Yaskawa INFORM job: A_ROOF_UPPER_0614_2_PAINT_55.JBI

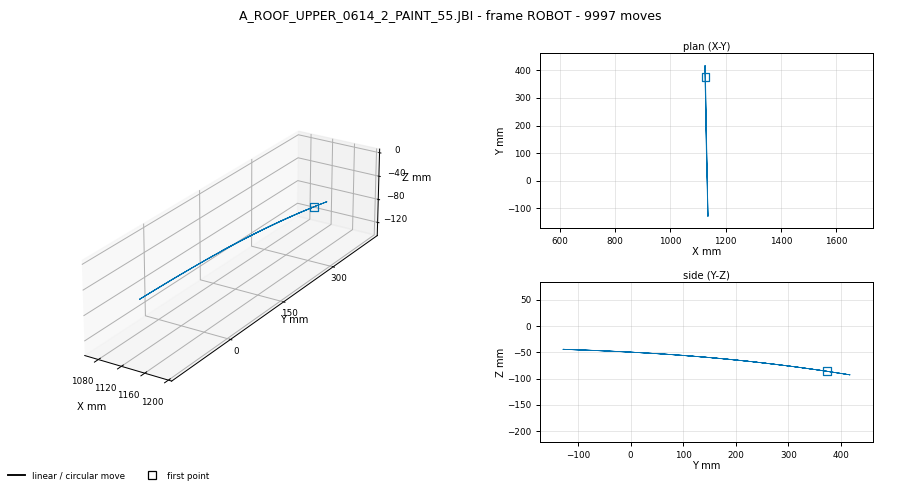
[picture p0: tool path of A_ROOF_UPPER_0614_2_PAINT_55.JBI in frame ROBOT, 9997 of 9997 moves have a stored position in this frame; points joined in program order, loops and branches not executed]
/JOB
//NAME A_ROOF_UPPER_0614_2_PAINT55
//POS
///NPOS 9997,0,0,0,0,0
///TOOL 1
///USER 0
///POSTYPE ROBOT
///RECTAN
///RCONF 1,0,0,0,0,0,0,0,0,0,0,0,0,0,0,0,0,0,0,0,0,0,0,0
C00000=1127.234,374.192,-85.938,-176.955,11.183,149.475
C00001=1127.238,373.945,-85.902,-176.958,11.180,149.475
C00002=1127.242,373.698,-85.865,-176.961,11.179,149.476
C00003=1127.246,373.451,-85.827,-176.964,11.176,149.476
C00004=1127.249,373.204,-85.790,-176.967,11.174,149.476
C00005=1127.253,372.957,-85.754,-176.971,11.171,149.476
C00006=1127.257,372.709,-85.717,-176.973,11.170,149.477
C00007=1127.261,372.462,-85.680,-176.976,11.167,149.477
C00008=1127.264,372.215,-85.643,-176.979,11.164,149.477
C00009=1127.268,371.968,-85.606,-176.983,11.162,149.477
C00010=1127.272,371.720,-85.570,-176.985,11.160,149.477
C00011=1127.276,371.473,-85.533,-176.989,11.158,149.477
C00012=1127.279,371.226,-85.496,-176.992,11.155,149.478
C00013=1127.283,370.978,-85.459,-176.995,11.153,149.478
C00014=1127.287,370.731,-85.423,-176.998,11.151,149.478
C00015=1127.291,370.484,-85.387,-177.001,11.149,149.478
C00016=1127.295,370.236,-85.350,-177.005,11.146,149.479
C00017=1127.299,369.989,-85.313,-177.008,11.144,149.479
C00018=1127.302,369.742,-85.276,-177.011,11.141,149.479
C00019=1127.306,369.495,-85.240,-177.014,11.139,149.479
C00020=1127.310,369.247,-85.203,-177.017,11.137,149.479
C00021=1127.313,369.000,-85.166,-177.020,11.134,149.480
C00022=1127.318,368.753,-85.130,-177.024,11.132,149.480
C00023=1127.321,368.506,-85.094,-177.027,11.130,149.480
C00024=1127.325,368.259,-85.057,-177.030,11.128,149.480
C00025=1127.329,368.011,-85.020,-177.033,11.125,149.480
C00026=1127.332,367.763,-84.984,-177.036,11.123,149.481
C00027=1127.336,367.516,-84.948,-177.040,11.120,149.481
C00028=1127.340,367.269,-84.911,-177.043,11.118,149.481
C00029=1127.344,367.022,-84.874,-177.046,11.115,149.481
C00030=1127.348,366.774,-84.839,-177.050,11.113,149.482
C00031=1127.352,366.527,-84.802,-177.053,11.112,149.482
C00032=1127.356,366.280,-84.765,-177.056,11.109,149.482
C00033=1127.359,366.033,-84.730,-177.059,11.107,149.482
C00034=1127.363,365.785,-84.693,-177.063,11.104,149.483
C00035=1127.367,365.538,-84.656,-177.066,11.102,149.483
C00036=1127.371,365.291,-84.620,-177.069,11.099,149.483
C00037=1127.374,365.043,-84.584,-177.072,11.097,149.483
C00038=1127.378,364.795,-84.548,-177.076,11.094,149.483
C00039=1127.382,364.548,-84.511,-177.079,11.092,149.484
C00040=1127.386,364.301,-84.474,-177.082,11.090,149.484
C00041=1127.390,364.054,-84.439,-177.085,11.088,149.484
C00042=1127.393,363.807,-84.403,-177.089,11.086,149.485
C00043=1127.397,363.559,-84.367,-177.092,11.083,149.485
C00044=1127.401,363.312,-84.330,-177.096,11.081,149.485
C00045=1127.405,363.064,-84.294,-177.099,11.078,149.485
C00046=1127.408,362.852,-84.263,-177.102,11.076,149.486
C00047=1127.412,362.640,-84.232,-177.105,11.074,149.486
C00048=1127.415,362.426,-84.201,-177.107,11.072,149.486
C00049=1127.418,362.214,-84.170,-177.111,11.070,149.486
C00050=1127.421,362.001,-84.139,-177.113,11.068,149.486
C00051=1127.425,361.789,-84.108,-177.117,11.066,149.487
C00052=1127.428,361.576,-84.077,-177.119,11.064,149.487
C00053=1127.431,361.363,-84.046,-177.122,11.062,149.487
C00054=1127.435,361.116,-84.010,-177.125,11.060,149.487
C00055=1127.438,360.869,-83.974,-177.129,11.057,149.488
C00056=1127.443,360.621,-83.938,-177.132,11.055,149.488
C00057=1127.446,360.374,-83.902,-177.136,11.052,149.488
C00058=1127.450,360.127,-83.866,-177.140,11.049,149.488
C00059=1127.453,359.879,-83.831,-177.143,11.047,149.489
C00060=1127.458,359.631,-83.795,-177.147,11.045,149.489
C00061=1127.461,359.384,-83.758,-177.150,11.042,149.489
C00062=1127.465,359.137,-83.723,-177.153,11.040,149.489
C00063=1127.470,358.890,-83.687,-177.156,11.037,149.490
C00064=1127.473,358.642,-83.651,-177.160,11.035,149.490
C00065=1127.477,358.395,-83.615,-177.163,11.033,149.490
C00066=1127.480,358.148,-83.580,-177.167,11.030,149.490
C00067=1127.485,357.900,-83.544,-177.170,11.028,149.491
C00068=1127.488,357.653,-83.508,-177.174,11.026,149.491
C00069=1127.492,357.405,-83.472,-177.177,11.023,149.491
C00070=1127.496,357.158,-83.437,-177.180,11.021,149.491
C00071=1127.499,356.910,-83.401,-177.184,11.018,149.492
C00072=1127.504,356.663,-83.364,-177.188,11.015,149.492
C00073=1127.508,356.416,-83.329,-177.191,11.013,149.492
C00074=1127.511,356.169,-83.294,-177.195,11.011,149.493
C00075=1127.515,355.921,-83.258,-177.198,11.008,149.493
C00076=1127.519,355.674,-83.223,-177.202,11.006,149.493
C00077=1127.522,355.426,-83.187,-177.206,11.003,149.493
C00078=1127.526,355.179,-83.152,-177.209,11.000,149.494
C00079=1127.531,354.932,-83.116,-177.212,10.998,149.494
C00080=1127.535,354.684,-83.080,-177.216,10.996,149.494
C00081=1127.538,354.437,-83.045,-177.219,10.993,149.494
C00082=1127.542,354.189,-83.009,-177.223,10.990,149.495
C00083=1127.546,353.941,-82.974,-177.227,10.988,149.495
C00084=1127.550,353.693,-82.939,-177.230,10.985,149.495
C00085=1127.554,353.447,-82.904,-177.233,10.983,149.495
C00086=1127.558,353.199,-82.868,-177.237,10.980,149.496
C00087=1127.561,352.952,-82.832,-177.241,10.978,149.496
C00088=1127.565,352.704,-82.797,-177.244,10.975,149.496
C00089=1127.569,352.457,-82.762,-177.248,10.973,149.497
C00090=1127.573,352.209,-82.727,-177.252,10.969,149.497
C00091=1127.577,351.962,-82.691,-177.255,10.967,149.497
C00092=1127.581,351.714,-82.656,-177.259,10.965,149.497
C00093=1127.585,351.467,-82.621,-177.262,10.962,149.498
C00094=1127.588,351.220,-82.585,-177.266,10.959,149.498
C00095=1127.592,350.972,-82.550,-177.269,10.957,149.498
C00096=1127.596,350.724,-82.515,-177.273,10.954,149.498
C00097=1127.600,350.478,-82.480,-177.277,10.951,149.499
C00098=1127.604,350.229,-82.445,-177.280,10.949,149.499
C00099=1127.608,349.982,-82.409,-177.284,10.946,149.499
C00100=1127.612,349.734,-82.374,-177.287,10.943,149.499
C00101=1127.616,349.487,-82.339,-177.291,10.941,149.500
C00102=1127.619,349.274,-82.309,-177.294,10.938,149.500
C00103=1127.623,349.061,-82.279,-177.297,10.936,149.500
C00104=1127.626,348.848,-82.248,-177.299,10.935,149.500
C00105=1127.629,348.636,-82.219,-177.302,10.932,149.500
C00106=1127.633,348.423,-82.188,-177.305,10.930,149.501
C00107=1127.636,348.210,-82.159,-177.308,10.928,149.501
C00108=1127.639,347.997,-82.128,-177.311,10.926,149.501
C00109=1127.643,347.785,-82.098,-177.313,10.924,149.501
C00110=1127.646,347.537,-82.063,-177.316,10.921,149.501
C00111=1127.651,347.290,-82.028,-177.320,10.919,149.501
C00112=1127.654,347.042,-81.993,-177.323,10.916,149.502
C00113=1127.658,346.794,-81.958,-177.326,10.914,149.502
C00114=1127.663,346.547,-81.923,-177.330,10.912,149.502
C00115=1127.667,346.299,-81.888,-177.333,10.909,149.502
C00116=1127.670,346.052,-81.853,-177.336,10.907,149.502
C00117=1127.674,345.805,-81.819,-177.339,10.904,149.503
C00118=1127.678,345.557,-81.784,-177.342,10.901,149.503
C00119=1127.682,345.310,-81.749,-177.346,10.899,149.503
C00120=1127.686,345.062,-81.714,-177.349,10.896,149.503
C00121=1127.690,344.814,-81.680,-177.352,10.894,149.503
C00122=1127.694,344.567,-81.644,-177.356,10.892,149.504
C00123=1127.698,344.319,-81.610,-177.359,10.889,149.504
C00124=1127.702,344.072,-81.576,-177.362,10.886,149.504
C00125=1127.705,343.824,-81.540,-177.365,10.884,149.504
C00126=1127.710,343.577,-81.506,-177.369,10.881,149.504
C00127=1127.714,343.329,-81.471,-177.372,10.879,149.505
C00128=1127.717,343.082,-81.436,-177.375,10.876,149.505
C00129=1127.721,342.834,-81.401,-177.378,10.874,149.505
C00130=1127.725,342.586,-81.367,-177.381,10.871,149.505
C00131=1127.729,342.339,-81.333,-177.385,10.869,149.505
C00132=1127.733,342.091,-81.298,-177.388,10.866,149.506
C00133=1127.737,341.844,-81.263,-177.391,10.865,149.506
C00134=1127.741,341.596,-81.228,-177.394,10.862,149.506
C00135=1127.745,341.349,-81.194,-177.397,10.860,149.506
C00136=1127.749,341.101,-81.159,-177.400,10.857,149.506
C00137=1127.753,340.854,-81.125,-177.404,10.854,149.507
C00138=1127.757,340.605,-81.090,-177.407,10.852,149.507
C00139=1127.761,340.358,-81.057,-177.410,10.850,149.507
C00140=1127.765,340.110,-81.022,-177.413,10.847,149.507
C00141=1127.769,339.863,-80.987,-177.416,10.844,149.507
C00142=1127.772,339.615,-80.953,-177.420,10.842,149.508
C00143=1127.777,339.368,-80.918,-177.423,10.839,149.508
C00144=1127.781,339.121,-80.884,-177.426,10.837,149.508
C00145=1127.785,338.873,-80.849,-177.430,10.835,149.508
C00146=1127.788,338.626,-80.815,-177.433,10.832,149.508
C00147=1127.793,338.377,-80.781,-177.436,10.829,149.509
C00148=1127.797,338.130,-80.747,-177.439,10.827,149.509
C00149=1127.800,337.882,-80.712,-177.443,10.824,149.509
C00150=1127.805,337.635,-80.678,-177.445,10.822,149.509
C00151=1127.808,337.387,-80.644,-177.449,10.819,149.509
C00152=1127.812,337.140,-80.610,-177.452,10.817,149.510
C00153=1127.817,336.892,-80.575,-177.455,10.814,149.510
C00154=1127.820,336.644,-80.541,-177.459,10.812,149.510
C00155=1127.824,336.397,-80.507,-177.462,10.809,149.510
C00156=1127.828,336.149,-80.472,-177.464,10.807,149.510
C00157=1127.832,335.902,-80.438,-177.468,10.805,149.511
C00158=1127.836,335.689,-80.409,-177.471,10.802,149.511
C00159=1127.839,335.475,-80.380,-177.473,10.800,149.511
C00160=1127.842,335.262,-80.351,-177.476,10.798,149.511
C00161=1127.845,335.050,-80.321,-177.479,10.796,149.511
C00162=1127.850,334.837,-80.292,-177.481,10.794,149.511
C00163=1127.853,334.623,-80.263,-177.484,10.792,149.512
C00164=1127.856,334.411,-80.233,-177.487,10.790,149.512
C00165=1127.859,334.198,-80.204,-177.490,10.787,149.512
C00166=1127.863,333.950,-80.170,-177.493,10.785,149.512
C00167=1127.867,333.702,-80.136,-177.497,10.782,149.512
C00168=1127.871,333.455,-80.102,-177.499,10.780,149.513
C00169=1127.875,333.207,-80.068,-177.502,10.778,149.513
C00170=1127.879,332.959,-80.034,-177.506,10.775,149.513
C00171=1127.883,332.712,-80.000,-177.509,10.773,149.513
C00172=1127.886,332.464,-79.966,-177.512,10.770,149.513
C00173=1127.891,332.216,-79.932,-177.515,10.768,149.514
C00174=1127.895,331.969,-79.899,-177.519,10.765,149.514
C00175=1127.898,331.721,-79.864,-177.521,10.762,149.514
C00176=1127.903,331.473,-79.831,-177.525,10.760,149.514
C00177=1127.907,331.226,-79.797,-177.528,10.757,149.514
C00178=1127.911,330.979,-79.764,-177.531,10.755,149.515
C00179=1127.914,330.731,-79.729,-177.534,10.752,149.515
C00180=1127.919,330.483,-79.696,-177.538,10.750,149.515
C00181=1127.923,330.236,-79.662,-177.541,10.747,149.515
C00182=1127.927,329.987,-79.628,-177.544,10.745,149.515
C00183=1127.931,329.740,-79.594,-177.547,10.742,149.515
C00184=1127.935,329.492,-79.561,-177.551,10.740,149.516
C00185=1127.939,329.245,-79.527,-177.554,10.737,149.516
C00186=1127.943,328.997,-79.493,-177.557,10.734,149.516
C00187=1127.947,328.749,-79.460,-177.560,10.732,149.516
C00188=1127.951,328.502,-79.426,-177.563,10.730,149.517
C00189=1127.955,328.254,-79.393,-177.566,10.728,149.517
C00190=1127.958,328.006,-79.359,-177.569,10.725,149.517
C00191=1127.963,327.758,-79.325,-177.572,10.723,149.517
C00192=1127.967,327.510,-79.292,-177.576,10.720,149.517
C00193=1127.971,327.263,-79.258,-177.579,10.717,149.517
C00194=1127.975,327.016,-79.225,-177.582,10.715,149.518
C00195=1127.979,326.767,-79.191,-177.585,10.713,149.518
C00196=1127.983,326.520,-79.157,-177.588,10.710,149.518
C00197=1127.987,326.272,-79.124,-177.592,10.707,149.518
C00198=1127.991,326.025,-79.091,-177.595,10.705,149.518
C00199=1127.995,325.777,-79.058,-177.598,10.702,149.518
C00200=1127.999,325.530,-79.024,-177.601,10.700,149.519
C00201=1128.002,325.281,-78.991,-177.604,10.697,149.519
C00202=1128.006,325.034,-78.957,-177.608,10.695,149.519
C00203=1128.011,324.786,-78.924,-177.611,10.692,149.519
C00204=1128.015,324.538,-78.891,-177.614,10.690,149.520
C00205=1128.019,324.291,-78.857,-177.617,10.687,149.520
C00206=1128.023,324.043,-78.824,-177.620,10.684,149.520
C00207=1128.027,323.795,-78.790,-177.624,10.682,149.520
C00208=1128.030,323.547,-78.757,-177.626,10.680,149.520
C00209=1128.034,323.299,-78.724,-177.629,10.677,149.520
C00210=1128.039,323.052,-78.691,-177.633,10.675,149.521
C00211=1128.043,322.804,-78.658,-177.636,10.673,149.521
C00212=1128.047,322.556,-78.625,-177.639,10.670,149.521
C00213=1128.051,322.308,-78.592,-177.642,10.667,149.521
C00214=1128.055,322.096,-78.563,-177.645,10.665,149.521
C00215=1128.058,321.883,-78.534,-177.648,10.663,149.522
C00216=1128.062,321.669,-78.506,-177.650,10.661,149.522
C00217=1128.064,321.456,-78.477,-177.653,10.658,149.522
C00218=1128.068,321.243,-78.448,-177.656,10.656,149.522
C00219=1128.071,321.030,-78.420,-177.659,10.654,149.522
C00220=1128.075,320.817,-78.391,-177.661,10.652,149.522
C00221=1128.078,320.603,-78.364,-177.664,10.650,149.522
C00222=1128.082,320.356,-78.330,-177.667,10.648,149.523
C00223=1128.086,320.108,-78.297,-177.670,10.645,149.523
C00224=1128.090,319.860,-78.264,-177.673,10.642,149.523
C00225=1128.095,319.613,-78.231,-177.676,10.640,149.523
C00226=1128.099,319.365,-78.198,-177.680,10.637,149.524
C00227=1128.102,319.117,-78.165,-177.683,10.635,149.524
C00228=1128.106,318.870,-78.132,-177.686,10.632,149.524
C00229=1128.111,318.621,-78.100,-177.689,10.629,149.524
C00230=1128.115,318.374,-78.066,-177.692,10.627,149.524
C00231=1128.119,318.126,-78.033,-177.696,10.625,149.524
C00232=1128.122,317.878,-78.001,-177.699,10.622,149.525
C00233=1128.127,317.631,-77.968,-177.702,10.619,149.525
C00234=1128.131,317.382,-77.935,-177.705,10.617,149.525
C00235=1128.135,317.135,-77.902,-177.708,10.614,149.525
C00236=1128.139,316.887,-77.869,-177.711,10.613,149.525
C00237=1128.143,316.639,-77.836,-177.714,10.610,149.525
C00238=1128.147,316.391,-77.804,-177.717,10.607,149.526
C00239=1128.151,316.144,-77.771,-177.720,10.605,149.526
C00240=1128.155,315.896,-77.738,-177.723,10.602,149.526
C00241=1128.159,315.648,-77.706,-177.727,10.600,149.526
C00242=1128.163,315.400,-77.673,-177.730,10.597,149.527
C00243=1128.167,315.152,-77.640,-177.733,10.594,149.527
C00244=1128.171,314.904,-77.608,-177.736,10.592,149.527
C00245=1128.175,314.656,-77.574,-177.739,10.589,149.527
C00246=1128.179,314.408,-77.543,-177.742,10.587,149.527
C00247=1128.183,314.161,-77.509,-177.746,10.584,149.527
C00248=1128.187,313.913,-77.476,-177.749,10.582,149.528
C00249=1128.191,313.665,-77.444,-177.752,10.579,149.528
C00250=1128.196,313.418,-77.412,-177.755,10.576,149.528
C00251=1128.199,313.170,-77.380,-177.758,10.574,149.528
C00252=1128.203,312.922,-77.347,-177.761,10.572,149.528
C00253=1128.208,312.674,-77.314,-177.764,10.569,149.528
C00254=1128.211,312.426,-77.282,-177.767,10.567,149.529
C00255=1128.216,312.178,-77.249,-177.770,10.564,149.529
C00256=1128.219,311.931,-77.217,-177.774,10.562,149.529
C00257=1128.224,311.682,-77.184,-177.777,10.559,149.529
C00258=1128.228,311.435,-77.153,-177.780,10.557,149.529
C00259=1128.232,311.187,-77.119,-177.783,10.554,149.530
C00260=1128.236,310.939,-77.087,-177.786,10.551,149.530
C00261=1128.240,310.691,-77.054,-177.789,10.549,149.530
C00262=1128.244,310.443,-77.022,-177.792,10.546,149.530
C00263=1128.248,310.195,-76.990,-177.796,10.544,149.530
C00264=1128.252,309.947,-76.957,-177.799,10.541,149.531
C00265=1128.256,309.700,-76.926,-177.802,10.539,149.531
C00266=1128.261,309.452,-76.893,-177.805,10.536,149.531
C00267=1128.264,309.204,-76.861,-177.808,10.533,149.531
C00268=1128.269,308.956,-76.828,-177.811,10.532,149.531
C00269=1128.272,308.708,-76.796,-177.814,10.529,149.531
C00270=1128.276,308.495,-76.769,-177.817,10.527,149.532
C00271=1128.280,308.282,-76.741,-177.819,10.525,149.532
C00272=1128.283,308.069,-76.713,-177.822,10.522,149.532
C00273=1128.287,307.855,-76.685,-177.825,10.520,149.532
C00274=1128.290,307.642,-76.658,-177.827,10.518,149.532
C00275=1128.293,307.429,-76.630,-177.831,10.516,149.532
C00276=1128.298,307.216,-76.602,-177.833,10.514,149.533
C00277=1128.301,307.002,-76.575,-177.835,10.512,149.533
C00278=1128.305,306.754,-76.542,-177.839,10.509,149.533
C00279=1128.309,306.506,-76.510,-177.842,10.506,149.533
C00280=1128.313,306.259,-76.479,-177.845,10.504,149.533
C00281=1128.318,306.011,-76.446,-177.848,10.501,149.533
C00282=1128.321,305.763,-76.415,-177.851,10.499,149.534
C00283=1128.325,305.514,-76.383,-177.854,10.496,149.534
C00284=1128.330,305.267,-76.351,-177.857,10.494,149.534
C00285=1128.334,305.019,-76.319,-177.861,10.491,149.534
C00286=1128.337,304.771,-76.287,-177.864,10.488,149.534
C00287=1128.342,304.523,-76.255,-177.867,10.486,149.535
C00288=1128.346,304.275,-76.223,-177.870,10.483,149.535
C00289=1128.350,304.027,-76.191,-177.873,10.481,149.535
C00290=1128.354,303.779,-76.159,-177.876,10.478,149.535
C00291=1128.359,303.531,-76.127,-177.879,10.476,149.535
C00292=1128.362,303.283,-76.095,-177.882,10.474,149.535
C00293=1128.366,303.035,-76.064,-177.885,10.471,149.536
C00294=1128.371,302.788,-76.032,-177.888,10.468,149.536
C00295=1128.375,302.540,-76.000,-177.891,10.466,149.536
C00296=1128.378,302.292,-75.968,-177.894,10.463,149.536
C00297=1128.383,302.044,-75.936,-177.898,10.461,149.536
C00298=1128.387,301.796,-75.904,-177.901,10.458,149.537
C00299=1128.392,301.549,-75.872,-177.904,10.456,149.537
C00300=1128.396,301.300,-75.841,-177.907,10.453,149.537
C00301=1128.399,301.052,-75.809,-177.910,10.450,149.537
C00302=1128.404,300.805,-75.778,-177.914,10.448,149.537
C00303=1128.408,300.556,-75.746,-177.916,10.445,149.537
C00304=1128.412,300.308,-75.714,-177.919,10.444,149.538
C00305=1128.416,300.060,-75.683,-177.922,10.441,149.538
C00306=1128.420,299.812,-75.651,-177.925,10.438,149.538
C00307=1128.424,299.565,-75.620,-177.928,10.436,149.538
C00308=1128.428,299.317,-75.588,-177.932,10.433,149.538
C00309=1128.432,299.068,-75.557,-177.935,10.430,149.538
C00310=1128.437,298.820,-75.525,-177.938,10.428,149.539
C00311=1128.441,298.572,-75.493,-177.941,10.425,149.539
C00312=1128.445,298.324,-75.462,-177.944,10.423,149.539
C00313=1128.449,298.076,-75.430,-177.947,10.420,149.539
C00314=1128.453,297.829,-75.399,-177.951,10.418,149.539
C00315=1128.457,297.580,-75.367,-177.953,10.415,149.540
C00316=1128.461,297.332,-75.336,-177.957,10.412,149.540
C00317=1128.465,297.085,-75.304,-177.959,10.410,149.540
C00318=1128.469,296.836,-75.273,-177.962,10.408,149.540
C00319=1128.474,296.589,-75.242,-177.965,10.405,149.540
C00320=1128.478,296.340,-75.210,-177.969,10.403,149.541
C00321=1128.482,296.093,-75.179,-177.972,10.400,149.541
C00322=1128.486,295.844,-75.148,-177.975,10.398,149.541
C00323=1128.490,295.597,-75.116,-177.978,10.395,149.541
C00324=1128.494,295.348,-75.085,-177.981,10.392,149.541
C00325=1128.499,295.101,-75.054,-177.984,10.390,149.541
C00326=1128.502,294.887,-75.027,-177.986,10.388,149.541
C00327=1128.506,294.673,-75.000,-177.990,10.385,149.542
C00328=1128.509,294.461,-74.973,-177.992,10.383,149.542
C00329=1128.513,294.247,-74.946,-177.994,10.381,149.542
C00330=1128.517,294.034,-74.919,-177.998,10.379,149.542
C00331=1128.520,293.820,-74.893,-178.000,10.377,149.542
C00332=1128.523,293.607,-74.865,-178.002,10.375,149.542
C00333=1128.527,293.394,-74.839,-178.005,10.372,149.542
C00334=1128.531,293.145,-74.807,-178.009,10.370,149.543
C00335=1128.536,292.897,-74.777,-178.012,10.367,149.543
C00336=1128.539,292.649,-74.745,-178.015,10.364,149.543
C00337=1128.543,292.402,-74.715,-178.017,10.362,149.543
C00338=1128.547,292.154,-74.683,-178.021,10.360,149.544
C00339=1128.552,291.906,-74.652,-178.023,10.357,149.544
C00340=1128.556,291.658,-74.621,-178.027,10.355,149.544
C00341=1128.560,291.409,-74.590,-178.030,10.352,149.544
C00342=1128.565,291.162,-74.559,-178.033,10.350,149.544
C00343=1128.568,290.913,-74.528,-178.036,10.347,149.544
C00344=1128.572,290.665,-74.497,-178.039,10.345,149.545
C00345=1128.576,290.417,-74.466,-178.042,10.342,149.545
C00346=1128.581,290.169,-74.435,-178.045,10.339,149.545
C00347=1128.585,289.921,-74.404,-178.049,10.337,149.545
C00348=1128.589,289.673,-74.373,-178.051,10.335,149.545
C00349=1128.593,289.425,-74.343,-178.054,10.332,149.545
C00350=1128.597,289.176,-74.312,-178.057,10.329,149.546
C00351=1128.602,288.929,-74.280,-178.060,10.327,149.546
C00352=1128.605,288.681,-74.250,-178.063,10.324,149.546
C00353=1128.609,288.433,-74.219,-178.067,10.322,149.546
C00354=1128.614,288.185,-74.188,-178.070,10.319,149.546
C00355=1128.619,287.937,-74.157,-178.073,10.317,149.547
C00356=1128.622,287.688,-74.127,-178.076,10.314,149.547
C00357=1128.627,287.441,-74.096,-178.079,10.311,149.547
C00358=1128.631,287.193,-74.065,-178.082,10.309,149.547
C00359=1128.634,286.944,-74.035,-178.085,10.307,149.547
C00360=1128.639,286.696,-74.004,-178.088,10.304,149.547
C00361=1128.644,286.448,-73.973,-178.091,10.301,149.548
C00362=1128.647,286.200,-73.943,-178.094,10.299,149.548
C00363=1128.652,285.952,-73.912,-178.097,10.296,149.548
C00364=1128.656,285.704,-73.881,-178.100,10.294,149.548
C00365=1128.659,285.456,-73.851,-178.103,10.291,149.548
C00366=1128.664,285.208,-73.820,-178.106,10.288,149.548
C00367=1128.668,284.960,-73.790,-178.110,10.286,149.549
C00368=1128.673,284.712,-73.759,-178.113,10.283,149.549
C00369=1128.677,284.463,-73.728,-178.115,10.282,149.549
C00370=1128.680,284.216,-73.698,-178.118,10.279,149.549
C00371=1128.685,283.968,-73.667,-178.122,10.276,149.549
C00372=1128.689,283.719,-73.637,-178.125,10.274,149.550
C00373=1128.693,283.471,-73.606,-178.127,10.271,149.550
C00374=1128.698,283.223,-73.575,-178.131,10.268,149.550
C00375=1128.702,282.975,-73.545,-178.134,10.266,149.550
C00376=1128.706,282.727,-73.514,-178.137,10.263,149.550
C00377=1128.710,282.478,-73.485,-178.140,10.260,149.550
C00378=1128.715,282.230,-73.454,-178.143,10.258,149.551
C00379=1128.718,281.983,-73.424,-178.146,10.256,149.551
C00380=1128.723,281.735,-73.393,-178.149,10.253,149.551
C00381=1128.727,281.486,-73.363,-178.152,10.251,149.551
C00382=1128.731,281.273,-73.337,-178.155,10.248,149.551
C00383=1128.734,281.060,-73.311,-178.158,10.246,149.552
C00384=1128.738,280.846,-73.285,-178.161,10.243,149.552
C00385=1128.742,280.632,-73.258,-178.165,10.241,149.552
C00386=1128.745,280.419,-73.233,-178.167,10.239,149.552
C00387=1128.749,280.205,-73.206,-178.170,10.236,149.552
C00388=1128.752,279.992,-73.181,-178.173,10.233,149.552
C00389=1128.756,279.778,-73.154,-178.176,10.231,149.553
C00390=1128.760,279.530,-73.125,-178.179,10.228,149.553
C00391=1128.764,279.282,-73.094,-178.183,10.226,149.553
C00392=1128.768,279.033,-73.064,-178.187,10.223,149.553
C00393=1128.773,278.785,-73.034,-178.190,10.220,149.553
C00394=1128.777,278.538,-73.003,-178.193,10.217,149.554
C00395=1128.781,278.290,-72.974,-178.197,10.214,149.554
C00396=1128.785,278.041,-72.943,-178.200,10.212,149.554
C00397=1128.789,277.793,-72.913,-178.203,10.209,149.554
C00398=1128.793,277.545,-72.883,-178.207,10.206,149.554
C00399=1128.798,277.296,-72.853,-178.210,10.203,149.555
C00400=1128.802,277.049,-72.823,-178.213,10.200,149.555
C00401=1128.806,276.800,-72.794,-178.216,10.198,149.555
C00402=1128.810,276.552,-72.764,-178.219,10.195,149.555
C00403=1128.815,276.304,-72.733,-178.223,10.192,149.555
C00404=1128.819,276.056,-72.704,-178.226,10.189,149.555
C00405=1128.822,275.808,-72.673,-178.229,10.186,149.555
C00406=1128.827,275.559,-72.644,-178.232,10.184,149.556
C00407=1128.832,275.311,-72.614,-178.235,10.181,149.556
C00408=1128.835,275.063,-72.584,-178.238,10.178,149.556
C00409=1128.840,274.815,-72.554,-178.241,10.175,149.556
C00410=1128.844,274.567,-72.525,-178.244,10.173,149.556
C00411=1128.848,274.319,-72.494,-178.247,10.170,149.556
C00412=1128.853,274.070,-72.465,-178.250,10.168,149.557
C00413=1128.857,273.822,-72.435,-178.253,10.165,149.557
C00414=1128.861,273.574,-72.406,-178.256,10.162,149.557
C00415=1128.865,273.326,-72.375,-178.259,10.160,149.557
C00416=1128.869,273.078,-72.346,-178.262,10.157,149.557
C00417=1128.874,272.829,-72.316,-178.265,10.154,149.557
C00418=1128.878,272.581,-72.287,-178.268,10.151,149.557
C00419=1128.882,272.333,-72.257,-178.271,10.149,149.557
C00420=1128.886,272.085,-72.227,-178.274,10.146,149.558
C00421=1128.890,271.837,-72.197,-178.277,10.143,149.558
C00422=1128.895,271.589,-72.168,-178.280,10.140,149.558
C00423=1128.899,271.340,-72.139,-178.283,10.138,149.558
C00424=1128.903,271.092,-72.109,-178.285,10.136,149.558
C00425=1128.908,270.844,-72.079,-178.288,10.133,149.558
C00426=1128.912,270.595,-72.050,-178.292,10.130,149.558
C00427=1128.916,270.347,-72.020,-178.295,10.128,149.558
C00428=1128.920,270.099,-71.991,-178.297,10.125,149.559
C00429=1128.924,269.851,-71.961,-178.299,10.123,149.559
C00430=1128.928,269.603,-71.931,-178.302,10.120,149.559
C00431=1128.933,269.355,-71.902,-178.305,10.117,149.559
C00432=1128.937,269.106,-71.872,-178.308,10.115,149.559
C00433=1128.941,268.858,-71.843,-178.310,10.112,149.559
C00434=1128.946,268.610,-71.814,-178.313,10.110,149.559
C00435=1128.950,268.362,-71.784,-178.316,10.108,149.559
C00436=1128.954,268.113,-71.755,-178.319,10.105,149.559
C00437=1128.959,267.865,-71.726,-178.321,10.103,149.559
C00438=1128.962,267.652,-71.701,-178.324,10.100,149.560
C00439=1128.966,267.438,-71.676,-178.326,10.098,149.560
C00440=1128.969,267.224,-71.649,-178.328,10.096,149.560
C00441=1128.973,267.010,-71.624,-178.330,10.094,149.560
C00442=1128.977,266.797,-71.599,-178.333,10.092,149.560
C00443=1128.980,266.583,-71.574,-178.335,10.090,149.560
C00444=1128.984,266.369,-71.549,-178.337,10.087,149.560
C00445=1128.988,266.156,-71.524,-178.339,10.085,149.560
C00446=1128.992,265.908,-71.495,-178.342,10.084,149.560
C00447=1128.996,265.659,-71.465,-178.344,10.082,149.560
C00448=1129.000,265.411,-71.436,-178.347,10.079,149.560
C00449=1129.004,265.163,-71.406,-178.349,10.076,149.560
C00450=1129.009,264.914,-71.378,-178.352,10.074,149.560
C00451=1129.014,264.666,-71.349,-178.354,10.072,149.561
C00452=1129.018,264.418,-71.319,-178.356,10.070,149.561
C00453=1129.022,264.170,-71.290,-178.360,10.067,149.561
C00454=1129.026,263.921,-71.261,-178.364,10.063,149.561
C00455=1129.030,263.673,-71.232,-178.368,10.060,149.562
C00456=1129.035,263.426,-71.203,-178.372,10.057,149.562
C00457=1129.039,263.177,-71.174,-178.376,10.053,149.562
C00458=1129.043,262.928,-71.145,-178.380,10.050,149.562
C00459=1129.047,262.680,-71.115,-178.383,10.048,149.562
C00460=1129.052,262.432,-71.086,-178.387,10.044,149.563
C00461=1129.056,262.184,-71.058,-178.391,10.041,149.563
C00462=1129.060,261.936,-71.029,-178.394,10.038,149.563
C00463=1129.065,261.687,-71.000,-178.398,10.035,149.563
C00464=1129.069,261.439,-70.971,-178.401,10.032,149.563
C00465=1129.073,261.191,-70.942,-178.405,10.029,149.564
C00466=1129.077,260.942,-70.913,-178.408,10.026,149.564
C00467=1129.082,260.694,-70.884,-178.411,10.023,149.564
C00468=1129.086,260.445,-70.855,-178.415,10.020,149.564
C00469=1129.090,260.198,-70.827,-178.419,10.016,149.564
C00470=1129.095,259.949,-70.798,-178.422,10.014,149.564
C00471=1129.099,259.701,-70.768,-178.425,10.011,149.565
C00472=1129.103,259.452,-70.740,-178.428,10.008,149.565
C00473=1129.108,259.204,-70.712,-178.431,10.005,149.565
C00474=1129.112,258.956,-70.682,-178.435,10.001,149.565
C00475=1129.116,258.707,-70.654,-178.438,9.999,149.565
C00476=1129.120,258.460,-70.625,-178.441,9.996,149.565
C00477=1129.125,258.211,-70.596,-178.444,9.993,149.565
C00478=1129.129,257.962,-70.568,-178.447,9.990,149.565
C00479=1129.133,257.715,-70.539,-178.450,9.987,149.565
C00480=1129.137,257.466,-70.511,-178.453,9.984,149.566
C00481=1129.142,257.217,-70.482,-178.456,9.981,149.566
C00482=1129.146,256.970,-70.453,-178.459,9.979,149.566
C00483=1129.150,256.721,-70.425,-178.462,9.976,149.566
C00484=1129.155,256.472,-70.396,-178.465,9.973,149.566
C00485=1129.159,256.225,-70.368,-178.468,9.970,149.566
C00486=1129.163,255.976,-70.339,-178.471,9.967,149.566
C00487=1129.167,255.727,-70.311,-178.471,9.966,149.566
C00488=1129.172,255.479,-70.283,-178.470,9.965,149.565
C00489=1129.175,255.231,-70.254,-178.469,9.965,149.565
C00490=1129.181,254.983,-70.225,-178.469,9.963,149.565
C00491=1129.184,254.735,-70.197,-178.470,9.962,149.565
C00492=1129.189,254.486,-70.169,-178.470,9.961,149.564
C00493=1129.194,254.237,-70.140,-178.470,9.960,149.564
C00494=1129.197,254.024,-70.116,-178.472,9.959,149.564
C00495=1129.201,253.810,-70.091,-178.472,9.958,149.564
C00496=1129.204,253.596,-70.067,-178.474,9.957,149.564
C00497=1129.208,253.382,-70.042,-178.475,9.955,149.564
C00498=1129.212,253.169,-70.017,-178.476,9.953,149.564
C00499=1129.215,252.955,-69.993,-178.478,9.951,149.564
C00500=1129.219,252.741,-69.969,-178.480,9.950,149.564
C00501=1129.223,252.527,-69.944,-178.482,9.948,149.564
C00502=1129.227,252.280,-69.916,-178.485,9.945,149.564
C00503=1129.231,252.031,-69.887,-178.488,9.944,149.565
C00504=1129.235,251.782,-69.859,-178.491,9.941,149.565
C00505=1129.240,251.534,-69.830,-178.495,9.938,149.565
C00506=1129.244,251.285,-69.802,-178.497,9.935,149.565
C00507=1129.249,251.037,-69.774,-178.501,9.932,149.566
C00508=1129.253,250.789,-69.746,-178.506,9.929,149.566
C00509=1129.258,250.541,-69.717,-178.511,9.925,149.566
C00510=1129.262,250.292,-69.689,-178.515,9.922,149.567
C00511=1129.265,250.043,-69.661,-178.520,9.918,149.567
C00512=1129.270,249.795,-69.633,-178.525,9.914,149.568
C00513=1129.274,249.547,-69.605,-178.530,9.910,149.568
C00514=1129.279,249.298,-69.576,-178.536,9.905,149.568
C00515=1129.283,249.050,-69.548,-178.541,9.901,149.569
C00516=1129.287,248.802,-69.520,-178.548,9.896,149.569
C00517=1129.291,248.553,-69.492,-178.554,9.892,149.570
C00518=1129.296,248.305,-69.464,-178.560,9.887,149.570
C00519=1129.300,248.057,-69.436,-178.567,9.881,149.571
C00520=1129.305,247.808,-69.409,-178.574,9.876,149.572
C00521=1129.309,247.560,-69.381,-178.581,9.871,149.572
C00522=1129.313,247.311,-69.352,-178.586,9.867,149.572
C00523=1129.318,247.063,-69.324,-178.587,9.864,149.572
C00524=1129.322,246.814,-69.297,-178.588,9.862,149.572
C00525=1129.326,246.566,-69.269,-178.589,9.860,149.572
C00526=1129.330,246.319,-69.241,-178.591,9.858,149.571
C00527=1129.335,246.069,-69.213,-178.592,9.856,149.571
C00528=1129.340,245.821,-69.186,-178.593,9.854,149.571
C00529=1129.343,245.573,-69.157,-178.595,9.852,149.571
C00530=1129.348,245.324,-69.130,-178.596,9.849,149.571
C00531=1129.352,245.076,-69.103,-178.597,9.848,149.571
C00532=1129.356,244.828,-69.074,-178.599,9.845,149.571
C00533=1129.362,244.579,-69.047,-178.601,9.843,149.571
C00534=1129.365,244.330,-69.019,-178.602,9.841,149.570
C00535=1129.370,244.082,-68.991,-178.604,9.839,149.570
C00536=1129.374,243.834,-68.964,-178.606,9.836,149.570
C00537=1129.378,243.585,-68.936,-178.608,9.834,149.570
C00538=1129.383,243.337,-68.909,-178.609,9.833,149.570
C00539=1129.387,243.089,-68.881,-178.611,9.830,149.570
C00540=1129.391,242.840,-68.853,-178.613,9.828,149.570
C00541=1129.396,242.592,-68.825,-178.615,9.826,149.570
C00542=1129.400,242.343,-68.797,-178.617,9.823,149.570
C00543=1129.405,242.094,-68.770,-178.618,9.821,149.570
C00544=1129.409,241.847,-68.742,-178.621,9.819,149.570
C00545=1129.413,241.597,-68.715,-178.623,9.817,149.570
C00546=1129.417,241.350,-68.687,-178.625,9.814,149.570
C00547=1129.422,241.101,-68.660,-178.626,9.812,149.570
C00548=1129.426,240.852,-68.632,-178.629,9.809,149.570
C00549=1129.430,240.604,-68.605,-178.631,9.807,149.570
C00550=1129.434,240.390,-68.581,-178.634,9.805,149.570
C00551=1129.438,240.176,-68.557,-178.635,9.803,149.570
C00552=1129.441,239.963,-68.533,-178.637,9.801,149.570
C00553=1129.446,239.748,-68.510,-178.639,9.799,149.570
C00554=1129.449,239.535,-68.486,-178.641,9.797,149.570
C00555=1129.453,239.321,-68.462,-178.643,9.795,149.570
C00556=1129.457,239.106,-68.439,-178.645,9.792,149.570
C00557=1129.460,238.893,-68.415,-178.647,9.790,149.570
C00558=1129.464,238.644,-68.388,-178.650,9.788,149.571
C00559=1129.469,238.396,-68.361,-178.652,9.785,149.570
C00560=1129.473,238.148,-68.333,-178.655,9.783,149.571
C00561=1129.478,237.899,-68.305,-178.658,9.781,149.571
C00562=1129.482,237.650,-68.278,-178.660,9.778,149.571
C00563=1129.487,237.402,-68.251,-178.662,9.776,149.571
C00564=1129.491,237.154,-68.223,-178.665,9.773,149.571
C00565=1129.495,236.905,-68.196,-178.668,9.770,149.571
C00566=1129.500,236.657,-68.168,-178.671,9.767,149.571
C00567=1129.504,236.408,-68.141,-178.674,9.765,149.571
C00568=1129.509,236.160,-68.114,-178.677,9.762,149.571
C00569=1129.514,235.911,-68.087,-178.679,9.759,149.571
C00570=1129.517,235.663,-68.060,-178.682,9.757,149.571
C00571=1129.521,235.414,-68.032,-178.685,9.754,149.572
C00572=1129.526,235.166,-68.005,-178.689,9.750,149.572
C00573=1129.531,234.917,-67.978,-178.691,9.748,149.572
C00574=1129.535,234.668,-67.951,-178.694,9.745,149.572
C00575=1129.539,234.420,-67.923,-178.697,9.742,149.572
C00576=1129.544,234.172,-67.896,-178.701,9.740,149.572
C00577=1129.548,233.924,-67.870,-178.704,9.737,149.573
C00578=1129.552,233.675,-67.843,-178.707,9.734,149.573
C00579=1129.556,233.426,-67.815,-178.710,9.731,149.573
C00580=1129.561,233.178,-67.788,-178.714,9.727,149.573
C00581=1129.565,232.929,-67.762,-178.717,9.725,149.573
C00582=1129.569,232.681,-67.735,-178.720,9.721,149.573
C00583=1129.574,232.432,-67.707,-178.723,9.718,149.573
C00584=1129.579,232.184,-67.680,-178.727,9.715,149.574
C00585=1129.583,231.935,-67.653,-178.730,9.712,149.574
C00586=1129.587,231.686,-67.627,-178.734,9.709,149.574
C00587=1129.591,231.438,-67.599,-178.737,9.705,149.574
C00588=1129.596,231.189,-67.572,-178.740,9.703,149.574
C00589=1129.600,230.941,-67.546,-178.744,9.699,149.574
C00590=1129.605,230.693,-67.519,-178.748,9.696,149.574
C00591=1129.609,230.444,-67.492,-178.751,9.692,149.575
C00592=1129.613,230.196,-67.465,-178.755,9.689,149.575
C00593=1129.618,229.948,-67.438,-178.759,9.686,149.575
C00594=1129.623,229.699,-67.411,-178.763,9.682,149.575
C00595=1129.626,229.451,-67.385,-178.766,9.679,149.575
C00596=1129.631,229.202,-67.358,-178.770,9.675,149.575
C00597=1129.636,228.953,-67.331,-178.774,9.672,149.576
C00598=1129.639,228.704,-67.304,-178.777,9.668,149.576
C00599=1129.644,228.456,-67.277,-178.781,9.665,149.576
C00600=1129.648,228.208,-67.251,-178.785,9.661,149.576
C00601=1129.653,227.959,-67.225,-178.788,9.658,149.576
C00602=1129.657,227.710,-67.198,-178.792,9.654,149.576
C00603=1129.662,227.462,-67.171,-178.795,9.651,149.576
C00604=1129.666,227.213,-67.145,-178.798,9.647,149.576
C00605=1129.670,226.965,-67.118,-178.802,9.643,149.576
C00606=1129.674,226.751,-67.095,-178.805,9.641,149.577
C00607=1129.678,226.537,-67.072,-178.808,9.638,149.577
C00608=1129.682,226.323,-67.050,-178.810,9.635,149.577
C00609=1129.686,226.109,-67.027,-178.813,9.632,149.577
C00610=1129.690,225.894,-67.004,-178.816,9.629,149.577
C00611=1129.694,225.681,-66.982,-178.819,9.626,149.577
C00612=1129.697,225.466,-66.958,-178.821,9.623,149.577
C00613=1129.701,225.253,-66.936,-178.824,9.620,149.577
C00614=1129.705,225.004,-66.910,-178.828,9.617,149.577
C00615=1129.710,224.755,-66.883,-178.830,9.614,149.577
C00616=1129.714,224.507,-66.857,-178.834,9.610,149.577
C00617=1129.718,224.258,-66.831,-178.837,9.607,149.577
C00618=1129.723,224.009,-66.804,-178.840,9.603,149.577
C00619=1129.727,223.761,-66.778,-178.843,9.601,149.577
C00620=1129.732,223.512,-66.751,-178.846,9.597,149.577
C00621=1129.737,223.265,-66.725,-178.848,9.594,149.577
C00622=1129.741,223.016,-66.700,-178.852,9.590,149.577
C00623=1129.746,222.767,-66.673,-178.855,9.587,149.577
C00624=1129.750,222.518,-66.647,-178.857,9.584,149.577
C00625=1129.754,222.270,-66.621,-178.860,9.580,149.577
C00626=1129.759,222.021,-66.594,-178.863,9.577,149.577
C00627=1129.763,221.772,-66.568,-178.865,9.574,149.577
C00628=1129.767,221.524,-66.542,-178.868,9.571,149.577
C00629=1129.772,221.276,-66.516,-178.870,9.568,149.577
C00630=1129.777,221.027,-66.490,-178.874,9.564,149.577
C00631=1129.781,220.778,-66.464,-178.876,9.561,149.577
C00632=1129.785,220.530,-66.438,-178.879,9.558,149.577
C00633=1129.790,220.281,-66.411,-178.881,9.554,149.576
C00634=1129.794,220.032,-66.386,-178.884,9.551,149.576
C00635=1129.799,219.784,-66.360,-178.886,9.548,149.576
C00636=1129.803,219.536,-66.334,-178.889,9.545,149.576
C00637=1129.808,219.287,-66.307,-178.891,9.542,149.576
C00638=1129.812,219.038,-66.282,-178.894,9.539,149.576
C00639=1129.816,218.789,-66.256,-178.896,9.536,149.576
C00640=1129.820,218.540,-66.230,-178.898,9.533,149.576
C00641=1129.825,218.293,-66.204,-178.900,9.530,149.576
C00642=1129.830,218.044,-66.178,-178.903,9.527,149.576
C00643=1129.834,217.795,-66.152,-178.905,9.524,149.576
C00644=1129.838,217.546,-66.126,-178.907,9.521,149.575
C00645=1129.843,217.298,-66.101,-178.909,9.518,149.575
C00646=1129.847,217.049,-66.075,-178.912,9.515,149.575
C00647=1129.851,216.800,-66.049,-178.913,9.512,149.575
C00648=1129.856,216.551,-66.023,-178.916,9.509,149.575
C00649=1129.861,216.302,-65.997,-178.918,9.507,149.575
C00650=1129.865,216.055,-65.971,-178.920,9.503,149.575
C00651=1129.869,215.806,-65.945,-178.922,9.501,149.574
C00652=1129.874,215.557,-65.920,-178.924,9.497,149.574
C00653=1129.878,215.308,-65.894,-178.926,9.495,149.574
C00654=1129.883,215.060,-65.869,-178.928,9.493,149.574
C00655=1129.887,214.812,-65.843,-178.930,9.489,149.574
C00656=1129.891,214.563,-65.817,-178.932,9.487,149.574
C00657=1129.896,214.315,-65.792,-178.933,9.484,149.574
C00658=1129.901,214.066,-65.765,-178.936,9.481,149.574
C00659=1129.905,213.817,-65.740,-178.937,9.478,149.573
C00660=1129.909,213.568,-65.714,-178.939,9.476,149.573
C00661=1129.914,213.320,-65.688,-178.940,9.473,149.573
C00662=1129.917,213.105,-65.667,-178.941,9.471,149.573
C00663=1129.922,212.891,-65.644,-178.943,9.469,149.573
C00664=1129.925,212.677,-65.623,-178.944,9.467,149.572
C00665=1129.930,212.463,-65.601,-178.946,9.465,149.572
C00666=1129.934,212.249,-65.578,-178.947,9.462,149.572
C00667=1129.937,212.034,-65.556,-178.949,9.461,149.572
C00668=1129.941,211.820,-65.534,-178.951,9.458,149.572
C00669=1129.945,211.606,-65.513,-178.951,9.456,149.572
C00670=1129.949,211.357,-65.487,-178.954,9.453,149.572
C00671=1129.954,211.109,-65.462,-178.956,9.451,149.572
C00672=1129.958,210.860,-65.436,-178.958,9.449,149.572
C00673=1129.962,210.612,-65.410,-178.960,9.446,149.572
C00674=1129.967,210.363,-65.385,-178.961,9.443,149.571
C00675=1129.971,210.114,-65.360,-178.963,9.441,149.571
C00676=1129.976,209.865,-65.334,-178.965,9.438,149.571
C00677=1129.980,209.617,-65.309,-178.967,9.436,149.571
C00678=1129.985,209.368,-65.283,-178.970,9.434,149.571
C00679=1129.989,209.119,-65.258,-178.972,9.431,149.571
C00680=1129.994,208.871,-65.232,-178.974,9.428,149.571
C00681=1129.998,208.622,-65.207,-178.977,9.425,149.571
C00682=1130.003,208.374,-65.181,-178.979,9.423,149.571
C00683=1130.007,208.125,-65.156,-178.981,9.420,149.571
C00684=1130.012,207.876,-65.130,-178.983,9.418,149.571
C00685=1130.017,207.628,-65.105,-178.986,9.415,149.571
C00686=1130.020,207.379,-65.080,-178.989,9.412,149.571
C00687=1130.025,207.130,-65.055,-178.991,9.410,149.571
C00688=1130.029,206.882,-65.030,-178.994,9.407,149.572
C00689=1130.034,206.633,-65.004,-178.996,9.404,149.572
C00690=1130.039,206.384,-64.979,-178.999,9.401,149.572
C00691=1130.043,206.135,-64.953,-179.002,9.398,149.572
C00692=1130.048,205.887,-64.928,-179.004,9.396,149.572
C00693=1130.052,205.638,-64.904,-179.007,9.393,149.572
C00694=1130.057,205.390,-64.878,-179.010,9.390,149.572
C00695=1130.061,205.140,-64.853,-179.012,9.387,149.572
C00696=1130.066,204.892,-64.828,-179.015,9.385,149.572
C00697=1130.070,204.643,-64.803,-179.019,9.381,149.572
C00698=1130.074,204.395,-64.778,-179.022,9.378,149.572
C00699=1130.079,204.146,-64.752,-179.024,9.375,149.572
C00700=1130.083,203.897,-64.727,-179.027,9.373,149.573
C00701=1130.088,203.649,-64.702,-179.030,9.370,149.573
C00702=1130.093,203.399,-64.677,-179.034,9.366,149.573
C00703=1130.097,203.152,-64.652,-179.037,9.364,149.573
C00704=1130.101,202.902,-64.627,-179.040,9.361,149.573
C00705=1130.106,202.653,-64.602,-179.043,9.357,149.573
C00706=1130.110,202.405,-64.577,-179.046,9.355,149.573
C00707=1130.115,202.156,-64.552,-179.050,9.351,149.574
C00708=1130.119,201.907,-64.527,-179.053,9.348,149.574
C00709=1130.124,201.659,-64.503,-179.057,9.345,149.574
C00710=1130.129,201.410,-64.478,-179.060,9.341,149.574
C00711=1130.133,201.161,-64.452,-179.063,9.339,149.574
C00712=1130.137,200.913,-64.428,-179.067,9.335,149.574
C00713=1130.142,200.664,-64.403,-179.070,9.331,149.574
C00714=1130.147,200.416,-64.378,-179.074,9.328,149.575
C00715=1130.150,200.166,-64.353,-179.077,9.324,149.575
C00716=1130.156,199.918,-64.329,-179.081,9.321,149.575
C00717=1130.159,199.669,-64.304,-179.085,9.317,149.575
C00718=1130.164,199.454,-64.282,-179.088,9.315,149.575
C00719=1130.167,199.240,-64.261,-179.090,9.312,149.575
C00720=1130.171,199.026,-64.240,-179.094,9.308,149.575
C00721=1130.175,198.812,-64.218,-179.097,9.306,149.576
C00722=1130.179,198.597,-64.198,-179.101,9.302,149.576
C00723=1130.183,198.384,-64.176,-179.104,9.299,149.576
C00724=1130.188,198.169,-64.155,-179.107,9.296,149.576
C00725=1130.191,197.955,-64.134,-179.110,9.293,149.576
C00726=1130.195,197.706,-64.109,-179.114,9.289,149.576
C00727=1130.200,197.457,-64.084,-179.118,9.285,149.576
C00728=1130.205,197.209,-64.060,-179.122,9.281,149.577
C00729=1130.209,196.959,-64.035,-179.126,9.278,149.577
C00730=1130.214,196.711,-64.011,-179.130,9.273,149.577
C00731=1130.218,196.463,-63.987,-179.134,9.270,149.577
C00732=1130.222,196.213,-63.962,-179.137,9.266,149.577
C00733=1130.227,195.965,-63.938,-179.139,9.264,149.577
C00734=1130.232,195.716,-63.913,-179.140,9.261,149.577
C00735=1130.236,195.467,-63.889,-179.142,9.259,149.577
C00736=1130.241,195.218,-63.864,-179.143,9.256,149.576
C00737=1130.245,194.970,-63.840,-179.145,9.253,149.576
C00738=1130.250,194.721,-63.816,-179.147,9.251,149.576
C00739=1130.254,194.472,-63.791,-179.148,9.248,149.576
C00740=1130.259,194.224,-63.767,-179.149,9.246,149.576
C00741=1130.263,193.975,-63.743,-179.151,9.244,149.576
C00742=1130.268,193.726,-63.718,-179.152,9.241,149.575
C00743=1130.272,193.477,-63.694,-179.154,9.239,149.575
C00744=1130.277,193.228,-63.670,-179.156,9.235,149.575
C00745=1130.282,192.980,-63.646,-179.158,9.233,149.575
C00746=1130.286,192.730,-63.621,-179.160,9.231,149.575
C00747=1130.291,192.482,-63.597,-179.162,9.228,149.575
C00748=1130.295,192.233,-63.573,-179.164,9.226,149.575
C00749=1130.299,191.985,-63.549,-179.165,9.223,149.574
C00750=1130.304,191.735,-63.524,-179.167,9.221,149.574
C00751=1130.309,191.486,-63.500,-179.169,9.218,149.574
C00752=1130.313,191.238,-63.476,-179.171,9.215,149.574
C00753=1130.317,190.990,-63.452,-179.173,9.212,149.574
C00754=1130.323,190.741,-63.427,-179.175,9.209,149.574
C00755=1130.327,190.491,-63.404,-179.177,9.207,149.574
C00756=1130.331,190.243,-63.380,-179.179,9.205,149.574
C00757=1130.336,189.994,-63.355,-179.182,9.202,149.574
C00758=1130.341,189.746,-63.331,-179.184,9.199,149.574
C00759=1130.345,189.497,-63.307,-179.186,9.196,149.574
C00760=1130.349,189.247,-63.283,-179.188,9.193,149.574
C00761=1130.354,188.999,-63.258,-179.190,9.190,149.574
C00762=1130.359,188.750,-63.234,-179.192,9.188,149.574
C00763=1130.363,188.501,-63.211,-179.194,9.185,149.574
C00764=1130.368,188.253,-63.187,-179.196,9.183,149.574
C00765=1130.372,188.004,-63.163,-179.199,9.180,149.573
C00766=1130.377,187.754,-63.138,-179.201,9.176,149.573
C00767=1130.381,187.506,-63.114,-179.203,9.174,149.573
C00768=1130.386,187.257,-63.091,-179.206,9.171,149.574
C00769=1130.390,187.009,-63.067,-179.209,9.168,149.573
C00770=1130.395,186.760,-63.043,-179.211,9.165,149.573
C00771=1130.400,186.511,-63.020,-179.213,9.163,149.573
C00772=1130.405,186.262,-62.995,-179.216,9.160,149.573
C00773=1130.409,186.013,-62.971,-179.218,9.157,149.573
C00774=1130.413,185.799,-62.951,-179.220,9.154,149.573
C00775=1130.416,185.584,-62.931,-179.223,9.151,149.573
C00776=1130.420,185.370,-62.910,-179.225,9.149,149.573
C00777=1130.424,185.155,-62.889,-179.228,9.146,149.573
C00778=1130.429,184.941,-62.869,-179.229,9.144,149.573
C00779=1130.433,184.727,-62.848,-179.231,9.141,149.573
C00780=1130.436,184.513,-62.828,-179.234,9.138,149.573
C00781=1130.440,184.298,-62.807,-179.236,9.136,149.573
C00782=1130.445,184.049,-62.784,-179.239,9.132,149.573
C00783=1130.449,183.801,-62.759,-179.242,9.129,149.573
C00784=1130.454,183.552,-62.736,-179.244,9.126,149.573
C00785=1130.458,183.303,-62.712,-179.247,9.124,149.573
C00786=1130.463,183.054,-62.689,-179.250,9.120,149.573
C00787=1130.467,182.805,-62.665,-179.253,9.117,149.573
C00788=1130.472,182.557,-62.641,-179.256,9.114,149.574
C00789=1130.477,182.308,-62.618,-179.259,9.111,149.574
C00790=1130.481,182.059,-62.595,-179.262,9.107,149.573
C00791=1130.486,181.810,-62.570,-179.265,9.104,149.574
C00792=1130.490,181.561,-62.547,-179.267,9.101,149.574
C00793=1130.495,181.312,-62.524,-179.270,9.097,149.574
C00794=1130.499,181.064,-62.500,-179.273,9.094,149.574
C00795=1130.504,180.815,-62.476,-179.276,9.090,149.574
C00796=1130.509,180.566,-62.453,-179.279,9.087,149.574
C00797=1130.514,180.317,-62.430,-179.283,9.084,149.574
C00798=1130.518,180.068,-62.406,-179.286,9.080,149.574
C00799=1130.523,179.819,-62.382,-179.289,9.077,149.574
C00800=1130.527,179.570,-62.359,-179.292,9.073,149.574
C00801=1130.532,179.321,-62.335,-179.295,9.069,149.574
C00802=1130.536,179.072,-62.313,-179.297,9.066,149.574
C00803=1130.540,178.824,-62.289,-179.299,9.064,149.574
C00804=1130.545,178.575,-62.265,-179.302,9.061,149.574
C00805=1130.550,178.326,-62.242,-179.304,9.057,149.573
C00806=1130.554,178.077,-62.219,-179.306,9.055,149.573
C00807=1130.559,177.828,-62.195,-179.308,9.052,149.573
C00808=1130.564,177.579,-62.172,-179.310,9.049,149.573
C00809=1130.568,177.330,-62.149,-179.312,9.046,149.573
C00810=1130.573,177.081,-62.126,-179.314,9.043,149.573
C00811=1130.577,176.832,-62.102,-179.316,9.040,149.573
C00812=1130.582,176.583,-62.079,-179.319,9.037,149.573
C00813=1130.586,176.335,-62.055,-179.321,9.034,149.573
C00814=1130.591,176.087,-62.033,-179.323,9.031,149.573
C00815=1130.596,175.837,-62.009,-179.325,9.028,149.572
C00816=1130.600,175.588,-61.986,-179.328,9.025,149.572
C00817=1130.605,175.339,-61.962,-179.329,9.023,149.572
C00818=1130.609,175.091,-61.940,-179.332,9.019,149.572
C00819=1130.614,174.842,-61.916,-179.334,9.016,149.572
C00820=1130.619,174.592,-61.894,-179.336,9.014,149.572
C00821=1130.623,174.343,-61.870,-179.338,9.011,149.572
C00822=1130.628,174.095,-61.848,-179.341,9.007,149.572
C00823=1130.633,173.846,-61.825,-179.342,9.005,149.572
C00824=1130.637,173.597,-61.801,-179.345,9.002,149.572
C00825=1130.641,173.348,-61.778,-179.347,8.998,149.572
C00826=1130.646,173.099,-61.755,-179.350,8.995,149.571
C00827=1130.651,172.850,-61.732,-179.351,8.993,149.571
C00828=1130.655,172.601,-61.709,-179.354,8.990,149.571
C00829=1130.660,172.353,-61.686,-179.357,8.986,149.571
C00830=1130.664,172.138,-61.666,-179.358,8.984,149.571
C00831=1130.668,171.924,-61.647,-179.360,8.981,149.571
C00832=1130.671,171.709,-61.627,-179.362,8.978,149.571
C00833=1130.676,171.494,-61.607,-179.364,8.976,149.571
C00834=1130.680,171.280,-61.588,-179.366,8.974,149.571
C00835=1130.684,171.065,-61.567,-179.369,8.971,149.571
C00836=1130.688,170.851,-61.548,-179.370,8.968,149.571
C00837=1130.691,170.636,-61.528,-179.372,8.966,149.571
C00838=1130.697,170.388,-61.505,-179.375,8.962,149.571
C00839=1130.702,170.138,-61.483,-179.377,8.959,149.570
C00840=1130.705,169.890,-61.460,-179.379,8.956,149.570
C00841=1130.710,169.641,-61.436,-179.382,8.953,149.570
C00842=1130.714,169.392,-61.414,-179.384,8.950,149.570
C00843=1130.720,169.143,-61.391,-179.386,8.947,149.570
C00844=1130.724,168.894,-61.368,-179.388,8.944,149.570
C00845=1130.728,168.645,-61.345,-179.391,8.941,149.570
C00846=1130.733,168.395,-61.323,-179.393,8.938,149.570
C00847=1130.738,168.147,-61.300,-179.396,8.934,149.570
C00848=1130.743,167.898,-61.277,-179.398,8.931,149.570
C00849=1130.747,167.649,-61.255,-179.400,8.928,149.570
C00850=1130.752,167.401,-61.232,-179.403,8.925,149.570
C00851=1130.757,167.151,-61.210,-179.405,8.922,149.569
C00852=1130.761,166.902,-61.186,-179.408,8.919,149.569
C00853=1130.765,166.654,-61.164,-179.410,8.915,149.569
C00854=1130.771,166.405,-61.141,-179.413,8.912,149.569
C00855=1130.775,166.156,-61.119,-179.415,8.909,149.569
C00856=1130.780,165.906,-61.096,-179.418,8.906,149.569
C00857=1130.784,165.658,-61.074,-179.420,8.902,149.569
C00858=1130.789,165.409,-61.052,-179.422,8.899,149.569
C00859=1130.793,165.160,-61.028,-179.425,8.896,149.569
C00860=1130.798,164.911,-61.006,-179.427,8.893,149.569
C00861=1130.803,164.662,-60.983,-179.430,8.890,149.569
C00862=1130.807,164.413,-60.961,-179.432,8.886,149.569
C00863=1130.812,164.164,-60.939,-179.434,8.883,149.568
C00864=1130.817,163.915,-60.916,-179.437,8.880,149.568
C00865=1130.821,163.666,-60.894,-179.439,8.877,149.568
C00866=1130.826,163.418,-60.872,-179.442,8.874,149.568
C00867=1130.831,163.168,-60.849,-179.444,8.870,149.568
C00868=1130.835,162.920,-60.827,-179.447,8.867,149.568
C00869=1130.839,162.671,-60.805,-179.449,8.864,149.568
C00870=1130.844,162.421,-60.782,-179.452,8.860,149.568
C00871=1130.849,162.173,-60.760,-179.454,8.857,149.568
C00872=1130.853,161.924,-60.737,-179.457,8.854,149.568
C00873=1130.858,161.674,-60.715,-179.459,8.851,149.568
C00874=1130.863,161.426,-60.693,-179.462,8.847,149.568
C00875=1130.867,161.177,-60.670,-179.464,8.844,149.567
C00876=1130.873,160.928,-60.648,-179.467,8.841,149.567
C00877=1130.877,160.679,-60.626,-179.470,8.837,149.567
C00878=1130.882,160.430,-60.604,-179.472,8.834,149.567
C00879=1130.886,160.181,-60.582,-179.474,8.830,149.567
C00880=1130.891,159.932,-60.559,-179.477,8.827,149.567
C00881=1130.896,159.683,-60.537,-179.480,8.823,149.567
C00882=1130.900,159.434,-60.515,-179.482,8.820,149.567
C00883=1130.905,159.185,-60.494,-179.485,8.817,149.567
C00884=1130.909,158.936,-60.471,-179.487,8.814,149.567
C00885=1130.914,158.687,-60.448,-179.490,8.810,149.567
C00886=1130.918,158.472,-60.430,-179.492,8.807,149.567
C00887=1130.922,158.258,-60.411,-179.494,8.804,149.567
C00888=1130.926,158.043,-60.392,-179.497,8.801,149.566
C00889=1130.930,157.828,-60.373,-179.498,8.798,149.566
C00890=1130.934,157.614,-60.354,-179.501,8.795,149.566
C00891=1130.938,157.399,-60.335,-179.503,8.792,149.566
C00892=1130.943,157.185,-60.316,-179.505,8.789,149.566
C00893=1130.946,156.970,-60.297,-179.507,8.786,149.566
C00894=1130.951,156.721,-60.275,-179.510,8.782,149.566
C00895=1130.955,156.472,-60.253,-179.513,8.779,149.566
C00896=1130.960,156.223,-60.231,-179.516,8.775,149.566
C00897=1130.964,155.974,-60.209,-179.518,8.772,149.566
C00898=1130.969,155.725,-60.188,-179.520,8.768,149.565
C00899=1130.974,155.477,-60.166,-179.523,8.764,149.565
C00900=1130.978,155.227,-60.144,-179.526,8.761,149.565
C00901=1130.983,154.979,-60.122,-179.529,8.757,149.565
C00902=1130.988,154.729,-60.100,-179.531,8.754,149.565
C00903=1130.993,154.480,-60.078,-179.534,8.750,149.565
C00904=1130.997,154.231,-60.056,-179.536,8.747,149.565
C00905=1131.002,153.982,-60.034,-179.540,8.743,149.565
C00906=1131.007,153.733,-60.013,-179.542,8.739,149.565
C00907=1131.012,153.484,-59.991,-179.545,8.735,149.565
C00908=1131.017,153.235,-59.970,-179.547,8.732,149.564
C00909=1131.021,152.986,-59.947,-179.550,8.728,149.564
C00910=1131.026,152.737,-59.926,-179.553,8.725,149.564
C00911=1131.031,152.488,-59.904,-179.555,8.721,149.564
C00912=1131.035,152.238,-59.883,-179.558,8.718,149.564
C00913=1131.039,151.990,-59.862,-179.561,8.713,149.564
C00914=1131.044,151.741,-59.840,-179.563,8.710,149.564
C00915=1131.048,151.492,-59.818,-179.566,8.706,149.563
C00916=1131.054,151.243,-59.797,-179.569,8.702,149.563
C00917=1131.058,150.994,-59.775,-179.571,8.699,149.563
C00918=1131.063,150.745,-59.753,-179.574,8.695,149.563
C00919=1131.068,150.496,-59.732,-179.577,8.690,149.563
C00920=1131.073,150.247,-59.711,-179.579,8.687,149.563
C00921=1131.077,149.998,-59.689,-179.582,8.683,149.563
C00922=1131.082,149.748,-59.668,-179.585,8.679,149.563
C00923=1131.086,149.500,-59.646,-179.587,8.676,149.562
C00924=1131.091,149.250,-59.625,-179.590,8.672,149.562
C00925=1131.096,149.001,-59.603,-179.593,8.667,149.562
C00926=1131.101,148.753,-59.582,-179.596,8.664,149.562
C00927=1131.106,148.504,-59.561,-179.598,8.660,149.562
C00928=1131.109,148.255,-59.539,-179.602,8.656,149.562
C00929=1131.115,148.005,-59.518,-179.604,8.652,149.562
C00930=1131.119,147.757,-59.497,-179.607,8.648,149.561
C00931=1131.125,147.507,-59.476,-179.610,8.645,149.561
C00932=1131.129,147.258,-59.454,-179.612,8.640,149.561
C00933=1131.133,147.009,-59.433,-179.615,8.636,149.561
C00934=1131.138,146.760,-59.412,-179.618,8.632,149.561
C00935=1131.143,146.511,-59.391,-179.621,8.628,149.561
C00936=1131.147,146.263,-59.370,-179.623,8.625,149.561
C00937=1131.152,146.013,-59.348,-179.626,8.621,149.560
C00938=1131.157,145.764,-59.327,-179.629,8.616,149.560
C00939=1131.162,145.515,-59.306,-179.631,8.612,149.560
C00940=1131.167,145.266,-59.285,-179.635,8.608,149.560
C00941=1131.172,145.017,-59.264,-179.637,8.604,149.560
C00942=1131.176,144.802,-59.246,-179.639,8.601,149.559
C00943=1131.179,144.587,-59.228,-179.640,8.598,149.559
C00944=1131.184,144.372,-59.209,-179.641,8.595,149.559
C00945=1131.187,144.157,-59.192,-179.642,8.592,149.558
C00946=1131.192,143.943,-59.173,-179.644,8.590,149.558
C00947=1131.195,143.728,-59.155,-179.644,8.587,149.558
C00948=1131.200,143.513,-59.137,-179.646,8.585,149.557
C00949=1131.204,143.299,-59.119,-179.647,8.581,149.557
C00950=1131.208,143.050,-59.098,-179.649,8.578,149.557
C00951=1131.213,142.801,-59.077,-179.650,8.575,149.556
C00952=1131.218,142.552,-59.056,-179.651,8.571,149.556
C00953=1131.223,142.303,-59.035,-179.653,8.568,149.556
C00954=1131.228,142.053,-59.014,-179.654,8.565,149.555
C00955=1131.232,141.804,-58.993,-179.656,8.562,149.555
C00956=1131.237,141.555,-58.972,-179.657,8.559,149.555
C00957=1131.241,141.306,-58.952,-179.658,8.555,149.554
C00958=1131.246,141.057,-58.931,-179.660,8.552,149.554
C00959=1131.251,140.808,-58.910,-179.662,8.548,149.554
C00960=1131.256,140.559,-58.889,-179.663,8.545,149.553
C00961=1131.260,140.310,-58.868,-179.664,8.542,149.553
C00962=1131.265,140.061,-58.847,-179.666,8.539,149.553
C00963=1131.269,139.812,-58.826,-179.667,8.536,149.552
C00964=1131.274,139.562,-58.806,-179.669,8.532,149.552
C00965=1131.279,139.313,-58.785,-179.670,8.529,149.552
C00966=1131.284,139.064,-58.764,-179.672,8.525,149.551
C00967=1131.288,138.815,-58.744,-179.673,8.523,149.551
C00968=1131.293,138.566,-58.722,-179.675,8.519,149.551
C00969=1131.298,138.318,-58.702,-179.676,8.516,149.550
C00970=1131.303,138.068,-58.681,-179.678,8.512,149.550
C00971=1131.307,137.819,-58.660,-179.679,8.509,149.550
C00972=1131.313,137.570,-58.639,-179.682,8.506,149.549
C00973=1131.317,137.321,-58.619,-179.683,8.503,149.549
C00974=1131.322,137.072,-58.598,-179.685,8.499,149.549
C00975=1131.327,136.823,-58.578,-179.686,8.496,149.548
C00976=1131.331,136.574,-58.557,-179.688,8.493,149.548
C00977=1131.336,136.325,-58.536,-179.689,8.490,149.548
C00978=1131.341,136.076,-58.516,-179.691,8.486,149.547
C00979=1131.346,135.826,-58.495,-179.692,8.483,149.547
C00980=1131.350,135.578,-58.475,-179.694,8.480,149.547
C00981=1131.355,135.329,-58.454,-179.695,8.477,149.547
C00982=1131.360,135.079,-58.433,-179.697,8.473,149.546
C00983=1131.364,134.830,-58.413,-179.698,8.470,149.546
C00984=1131.370,134.580,-58.393,-179.700,8.466,149.545
C00985=1131.374,134.332,-58.372,-179.701,8.464,149.545
C00986=1131.379,134.083,-58.352,-179.704,8.460,149.545
C00987=1131.384,133.833,-58.331,-179.705,8.457,149.545
C00988=1131.388,133.584,-58.311,-179.707,8.454,149.544
C00989=1131.393,133.335,-58.290,-179.708,8.451,149.544
C00990=1131.398,133.086,-58.269,-179.710,8.447,149.544
C00991=1131.402,132.837,-58.249,-179.712,8.444,149.543
C00992=1131.407,132.588,-58.229,-179.713,8.440,149.543
C00993=1131.412,132.338,-58.208,-179.715,8.437,149.543
C00994=1131.417,132.089,-58.188,-179.716,8.434,149.543
C00995=1131.421,131.840,-58.168,-179.718,8.430,149.542
C00996=1131.426,131.591,-58.147,-179.719,8.428,149.542
C00997=1131.431,131.342,-58.127,-179.721,8.424,149.542
C00998=1131.435,131.127,-58.109,-179.723,8.421,149.542
C00999=1131.439,130.912,-58.092,-179.724,8.418,149.541
C01000=1131.443,130.697,-58.074,-179.725,8.416,149.541
C01001=1131.448,130.483,-58.057,-179.727,8.413,149.541
C01002=1131.451,130.268,-58.039,-179.729,8.409,149.540
C01003=1131.456,130.053,-58.022,-179.730,8.407,149.540
C01004=1131.460,129.838,-58.004,-179.732,8.404,149.540
C01005=1131.464,129.623,-57.987,-179.733,8.401,149.540
C01006=1131.468,129.374,-57.966,-179.735,8.397,149.539
C01007=1131.473,129.125,-57.945,-179.736,8.395,149.539
C01008=1131.478,128.876,-57.926,-179.738,8.391,149.539
C01009=1131.483,128.627,-57.906,-179.740,8.389,149.539
C01010=1131.487,128.378,-57.885,-179.741,8.385,149.538
C01011=1131.492,128.129,-57.866,-179.743,8.381,149.538
C01012=1131.497,127.879,-57.845,-179.745,8.378,149.538
C01013=1131.502,127.630,-57.825,-179.747,8.375,149.538
C01014=1131.506,127.381,-57.805,-179.749,8.371,149.537
C01015=1131.511,127.132,-57.784,-179.750,8.368,149.537
C01016=1131.516,126.883,-57.765,-179.752,8.365,149.537
C01017=1131.521,126.634,-57.745,-179.754,8.361,149.536
C01018=1131.525,126.385,-57.725,-179.755,8.358,149.536
C01019=1131.531,126.135,-57.704,-179.757,8.355,149.536
C01020=1131.535,125.886,-57.684,-179.759,8.351,149.536
C01021=1131.540,125.637,-57.664,-179.761,8.349,149.535
C01022=1131.545,125.389,-57.644,-179.762,8.345,149.535
C01023=1131.550,125.139,-57.624,-179.764,8.341,149.535
C01024=1131.554,124.890,-57.604,-179.767,8.338,149.534
C01025=1131.559,124.640,-57.584,-179.768,8.335,149.534
C01026=1131.563,124.392,-57.564,-179.770,8.331,149.534
C01027=1131.568,124.142,-57.544,-179.772,8.328,149.534
C01028=1131.573,123.894,-57.524,-179.773,8.325,149.533
C01029=1131.578,123.644,-57.505,-179.775,8.321,149.533
C01030=1131.582,123.395,-57.485,-179.777,8.318,149.533
C01031=1131.587,123.146,-57.465,-179.779,8.314,149.533
C01032=1131.592,122.897,-57.445,-179.780,8.311,149.532
C01033=1131.597,122.648,-57.425,-179.782,8.308,149.532
C01034=1131.601,122.398,-57.405,-179.784,8.304,149.532
C01035=1131.606,122.149,-57.386,-179.787,8.301,149.532
C01036=1131.611,121.900,-57.366,-179.788,8.298,149.531
C01037=1131.616,121.651,-57.346,-179.790,8.294,149.531
C01038=1131.621,121.401,-57.326,-179.792,8.291,149.531
C01039=1131.625,121.152,-57.306,-179.794,8.287,149.531
C01040=1131.630,120.903,-57.287,-179.796,8.284,149.530
C01041=1131.635,120.654,-57.267,-179.797,8.281,149.530
C01042=1131.640,120.405,-57.247,-179.799,8.277,149.530
C01043=1131.644,120.155,-57.227,-179.801,8.274,149.529
C01044=1131.650,119.907,-57.208,-179.803,8.270,149.529
C01045=1131.654,119.658,-57.187,-179.805,8.267,149.529
C01046=1131.659,119.408,-57.168,-179.807,8.263,149.529
C01047=1131.664,119.159,-57.148,-179.808,8.260,149.528
C01048=1131.669,118.910,-57.129,-179.810,8.257,149.528
C01049=1131.673,118.661,-57.108,-179.812,8.253,149.528
C01050=1131.678,118.411,-57.089,-179.814,8.250,149.528
C01051=1131.683,118.163,-57.070,-179.816,8.246,149.527
C01052=1131.688,117.913,-57.050,-179.818,8.243,149.527
C01053=1131.692,117.663,-57.031,-179.819,8.239,149.527
C01054=1131.697,117.415,-57.011,-179.821,8.236,149.527
C01055=1131.702,117.167,-56.991,-179.824,8.232,149.526
C01056=1131.707,116.918,-56.972,-179.826,8.229,149.526
C01057=1131.711,116.670,-56.953,-179.828,8.225,149.526
C01058=1131.717,116.422,-56.933,-179.830,8.222,149.526
C01059=1131.721,116.174,-56.914,-179.831,8.218,149.525
C01060=1131.726,115.925,-56.895,-179.833,8.215,149.525
C01061=1131.730,115.677,-56.875,-179.835,8.211,149.525
C01062=1131.736,115.428,-56.856,-179.837,8.208,149.525
C01063=1131.741,115.178,-56.836,-179.839,8.205,149.524
C01064=1131.745,114.929,-56.817,-179.841,8.201,149.524
C01065=1131.751,114.680,-56.797,-179.843,8.198,149.524
C01066=1131.755,114.431,-56.778,-179.845,8.194,149.524
C01067=1131.759,114.181,-56.759,-179.847,8.191,149.523
C01068=1131.765,113.932,-56.739,-179.849,8.187,149.523
C01069=1131.770,113.683,-56.720,-179.851,8.184,149.523
C01070=1131.774,113.434,-56.701,-179.853,8.180,149.522
C01071=1131.779,113.185,-56.681,-179.855,8.176,149.522
C01072=1131.784,112.936,-56.662,-179.857,8.173,149.522
C01073=1131.788,112.686,-56.643,-179.859,8.169,149.522
C01074=1131.794,112.438,-56.624,-179.861,8.166,149.522
C01075=1131.798,112.188,-56.604,-179.863,8.162,149.521
C01076=1131.803,111.938,-56.584,-179.864,8.158,149.521
C01077=1131.808,111.690,-56.566,-179.867,8.155,149.521
C01078=1131.812,111.440,-56.546,-179.869,8.151,149.520
C01079=1131.818,111.191,-56.527,-179.871,8.148,149.520
C01080=1131.822,110.942,-56.508,-179.873,8.144,149.520
C01081=1131.827,110.693,-56.489,-179.875,8.140,149.520
C01082=1131.832,110.443,-56.469,-179.877,8.137,149.520
C01083=1131.837,110.195,-56.451,-179.880,8.132,149.519
C01084=1131.841,109.945,-56.431,-179.883,8.128,149.519
C01085=1131.846,109.696,-56.413,-179.886,8.124,149.519
C01086=1131.869,108.518,-56.325,-179.265,6.873,149.056
C01087=1131.874,108.282,-56.307,-179.267,6.872,149.057
C01088=1131.878,108.045,-56.290,-179.270,6.870,149.057
C01089=1131.883,107.809,-56.272,-179.272,6.869,149.058
C01090=1131.888,107.560,-56.254,-179.275,6.867,149.058
C01091=1131.894,107.310,-56.235,-179.278,6.865,149.058
C01092=1131.898,107.061,-56.216,-179.281,6.864,149.059
C01093=1131.902,106.812,-56.198,-179.283,6.862,149.059
C01094=1131.908,106.563,-56.179,-179.286,6.860,149.060
C01095=1131.912,106.313,-56.160,-179.289,6.859,149.060
C01096=1131.917,106.064,-56.142,-179.291,6.857,149.060
C01097=1131.922,105.815,-56.123,-179.294,6.855,149.061
C01098=1131.927,105.547,-56.104,-179.298,6.853,149.061
C01099=1131.932,105.278,-56.084,-179.301,6.851,149.062
C01100=1131.938,105.009,-56.064,-179.303,6.850,149.062
C01101=1131.943,104.742,-56.044,-179.306,6.848,149.063
C01102=1131.948,104.492,-56.025,-179.309,6.846,149.063
C01103=1131.953,104.243,-56.007,-179.312,6.845,149.064
C01104=1131.957,103.994,-55.988,-179.315,6.843,149.064
C01105=1131.962,103.745,-55.970,-179.318,6.842,149.065
C01106=1131.968,103.495,-55.952,-179.320,6.840,149.065
C01107=1131.973,103.246,-55.934,-179.323,6.838,149.065
C01108=1131.977,102.997,-55.914,-179.326,6.837,149.066
C01109=1131.981,102.747,-55.897,-179.329,6.835,149.066
C01110=1131.987,102.498,-55.878,-179.331,6.833,149.067
C01111=1131.992,102.249,-55.860,-179.334,6.832,149.067
C01112=1131.996,101.999,-55.842,-179.337,6.830,149.067
C01113=1132.001,101.750,-55.823,-179.340,6.828,149.068
C01114=1132.006,101.501,-55.805,-179.342,6.827,149.068
C01115=1132.012,101.252,-55.786,-179.345,6.825,149.069
C01116=1132.016,101.003,-55.768,-179.348,6.824,149.069
C01117=1132.021,100.753,-55.750,-179.351,6.822,149.070
C01118=1132.026,100.503,-55.732,-179.354,6.820,149.070
C01119=1132.031,100.254,-55.714,-179.356,6.819,149.071
C01120=1132.035,100.005,-55.696,-179.359,6.817,149.071
C01121=1132.040,99.757,-55.677,-179.362,6.815,149.071
C01122=1132.045,99.506,-55.658,-179.365,6.814,149.072
C01123=1132.050,99.257,-55.640,-179.367,6.812,149.072
C01124=1132.055,99.008,-55.622,-179.370,6.810,149.073
C01125=1132.060,98.759,-55.605,-179.373,6.809,149.073
C01126=1132.065,98.510,-55.587,-179.376,6.807,149.074
C01127=1132.070,98.261,-55.569,-179.379,6.806,149.074
C01128=1132.074,98.011,-55.550,-179.382,6.804,149.075
C01129=1132.079,97.761,-55.532,-179.384,6.803,149.075
C01130=1132.084,97.512,-55.514,-179.387,6.801,149.075
C01131=1132.089,97.263,-55.496,-179.390,6.799,149.076
C01132=1132.094,97.014,-55.478,-179.393,6.798,149.076
C01133=1132.099,96.765,-55.460,-179.395,6.796,149.077
C01134=1132.104,96.515,-55.442,-179.398,6.794,149.077
C01135=1132.109,96.266,-55.424,-179.401,6.793,149.077
C01136=1132.113,96.016,-55.405,-179.404,6.791,149.078
C01137=1132.119,95.766,-55.388,-179.406,6.790,149.079
C01138=1132.124,95.517,-55.370,-179.409,6.789,149.079
C01139=1132.128,95.268,-55.352,-179.412,6.787,149.079
C01140=1132.133,95.019,-55.334,-179.414,6.785,149.080
C01141=1132.138,94.770,-55.316,-179.417,6.784,149.080
C01142=1132.143,94.521,-55.298,-179.420,6.782,149.081
C01143=1132.148,94.271,-55.280,-179.423,6.780,149.081
C01144=1132.153,94.022,-55.262,-179.426,6.779,149.082
C01145=1132.158,93.773,-55.246,-179.429,6.777,149.082
C01146=1132.162,93.524,-55.228,-179.431,6.776,149.083
C01147=1132.167,93.274,-55.210,-179.434,6.774,149.083
C01148=1132.172,93.025,-55.192,-179.437,6.772,149.083
C01149=1132.177,92.775,-55.173,-179.440,6.771,149.084
C01150=1132.182,92.526,-55.156,-179.442,6.770,149.084
C01151=1132.187,92.276,-55.138,-179.444,6.768,149.085
C01152=1132.192,92.027,-55.120,-179.448,6.767,149.085
C01153=1132.197,91.778,-55.102,-179.450,6.765,149.086
C01154=1132.202,91.528,-55.085,-179.453,6.764,149.086
C01155=1132.207,91.279,-55.067,-179.456,6.762,149.087
C01156=1132.211,91.030,-55.050,-179.459,6.760,149.087
C01157=1132.216,90.781,-55.032,-179.461,6.759,149.087
C01158=1132.221,90.531,-55.014,-179.464,6.757,149.088
C01159=1132.226,90.282,-54.996,-179.467,6.756,149.088
C01160=1132.231,90.033,-54.978,-179.470,6.754,149.089
C01161=1132.236,89.783,-54.961,-179.472,6.753,149.089
C01162=1132.241,89.534,-54.943,-179.475,6.752,149.090
C01163=1132.245,89.284,-54.926,-179.478,6.750,149.090
C01164=1132.250,89.035,-54.908,-179.480,6.748,149.091
C01165=1132.255,88.786,-54.890,-179.483,6.747,149.091
C01166=1132.260,88.536,-54.873,-179.486,6.745,149.092
C01167=1132.265,88.287,-54.855,-179.489,6.744,149.092
C01168=1132.270,88.038,-54.839,-179.492,6.742,149.093
C01169=1132.275,87.789,-54.821,-179.494,6.741,149.093
C01170=1132.280,87.540,-54.803,-179.497,6.739,149.093
C01171=1132.285,87.290,-54.786,-179.500,6.738,149.094
C01172=1132.290,87.041,-54.768,-179.502,6.736,149.094
C01173=1132.295,86.791,-54.751,-179.506,6.735,149.095
C01174=1132.300,86.542,-54.733,-179.508,6.733,149.095
C01175=1132.305,86.292,-54.716,-179.511,6.732,149.096
C01176=1132.309,86.044,-54.698,-179.514,6.730,149.096
C01177=1132.314,85.794,-54.681,-179.516,6.729,149.097
C01178=1132.319,85.545,-54.663,-179.519,6.727,149.097
C01179=1132.324,85.295,-54.646,-179.522,6.726,149.098
C01180=1132.329,85.046,-54.628,-179.525,6.724,149.098
C01181=1132.334,84.797,-54.612,-179.527,6.723,149.098
C01182=1132.340,84.547,-54.594,-179.530,6.721,149.099
C01183=1132.344,84.298,-54.577,-179.533,6.720,149.099
C01184=1132.349,84.048,-54.560,-179.535,6.719,149.100
C01185=1132.354,83.799,-54.542,-179.538,6.717,149.100
C01186=1132.358,83.550,-54.525,-179.541,6.716,149.101
C01187=1132.364,83.300,-54.508,-179.544,6.714,149.101
C01188=1132.369,83.051,-54.490,-179.546,6.712,149.102
C01189=1132.374,82.802,-54.473,-179.549,6.711,149.102
C01190=1132.379,82.553,-54.455,-179.551,6.710,149.103
C01191=1132.383,82.303,-54.439,-179.555,6.709,149.103
C01192=1132.388,82.054,-54.422,-179.557,6.707,149.104
C01193=1132.393,81.804,-54.404,-179.560,6.705,149.104
C01194=1132.398,81.555,-54.387,-179.563,6.704,149.104
C01195=1132.404,81.306,-54.370,-179.566,6.702,149.105
C01196=1132.408,81.056,-54.353,-179.568,6.702,149.106
C01197=1132.413,80.807,-54.335,-179.571,6.700,149.106
C01198=1132.418,80.557,-54.318,-179.574,6.698,149.106
C01199=1132.423,80.308,-54.301,-179.576,6.697,149.107
C01200=1132.428,80.059,-54.285,-179.579,6.695,149.107
C01201=1132.433,79.810,-54.267,-179.582,6.693,149.108
C01202=1132.438,79.541,-54.248,-179.585,6.692,149.108
C01203=1132.443,79.273,-54.231,-179.588,6.690,149.109
C01204=1132.449,79.004,-54.212,-179.591,6.689,149.109
C01205=1132.454,78.735,-54.193,-179.594,6.687,149.110
C01206=1132.459,78.487,-54.177,-179.596,6.687,149.110
C01207=1132.464,78.237,-54.160,-179.599,6.685,149.111
C01208=1132.469,77.987,-54.143,-179.602,6.683,149.111
C01209=1132.474,77.738,-54.125,-179.605,6.682,149.112
C01210=1132.479,77.489,-54.109,-179.608,6.680,149.112
C01211=1132.484,77.240,-54.092,-179.610,6.679,149.113
C01212=1132.488,76.990,-54.075,-179.612,6.678,149.113
C01213=1132.493,76.741,-54.058,-179.615,6.676,149.114
C01214=1132.499,76.492,-54.041,-179.618,6.675,149.114
C01215=1132.503,76.242,-54.025,-179.621,6.673,149.115
C01216=1132.508,75.992,-54.007,-179.623,6.672,149.115
C01217=1132.513,75.743,-53.991,-179.626,6.671,149.115
C01218=1132.519,75.494,-53.974,-179.629,6.669,149.116
C01219=1132.523,75.244,-53.957,-179.632,6.668,149.117
C01220=1132.528,74.995,-53.940,-179.634,6.667,149.117
C01221=1132.534,74.746,-53.924,-179.637,6.665,149.117
C01222=1132.538,74.496,-53.907,-179.640,6.664,149.118
C01223=1132.543,74.246,-53.890,-179.642,6.662,149.118
C01224=1132.548,73.998,-53.873,-179.646,6.661,149.119
C01225=1132.553,73.748,-53.857,-179.648,6.660,149.119
C01226=1132.558,73.498,-53.839,-179.651,6.658,149.120
C01227=1132.563,73.250,-53.823,-179.653,6.657,149.120
C01228=1132.568,73.000,-53.806,-179.656,6.655,149.121
C01229=1132.573,72.750,-53.789,-179.659,6.654,149.121
C01230=1132.578,72.501,-53.773,-179.661,6.653,149.122
C01231=1132.582,72.252,-53.756,-179.664,6.651,149.122
C01232=1132.588,72.002,-53.739,-179.667,6.650,149.123
C01233=1132.593,71.753,-53.723,-179.670,6.649,149.123
C01234=1132.597,71.504,-53.706,-179.672,6.647,149.124
C01235=1132.602,71.254,-53.689,-179.675,6.646,149.124
C01236=1132.607,71.005,-53.672,-179.678,6.644,149.125
C01237=1132.612,70.755,-53.656,-179.680,6.643,149.125
C01238=1132.618,70.506,-53.640,-179.683,6.642,149.126
C01239=1132.623,70.257,-53.623,-179.686,6.640,149.126
C01240=1132.627,70.007,-53.606,-179.689,6.639,149.127
C01241=1132.632,69.758,-53.590,-179.691,6.638,149.127
C01242=1132.638,69.508,-53.573,-179.694,6.636,149.127
C01243=1132.642,69.258,-53.557,-179.697,6.635,149.128
C01244=1132.647,69.010,-53.540,-179.700,6.633,149.129
C01245=1132.652,68.760,-53.524,-179.702,6.632,149.129
C01246=1132.657,68.511,-53.507,-179.705,6.631,149.129
C01247=1132.662,68.261,-53.491,-179.708,6.630,149.130
C01248=1132.667,68.012,-53.475,-179.710,6.629,149.130
C01249=1132.672,67.763,-53.458,-179.713,6.627,149.131
C01250=1132.676,67.513,-53.441,-179.715,6.625,149.131
C01251=1132.682,67.264,-53.425,-179.719,6.624,149.132
C01252=1132.687,67.014,-53.408,-179.721,6.623,149.132
C01253=1132.692,66.765,-53.392,-179.724,6.622,149.133
C01254=1132.697,66.515,-53.376,-179.726,6.620,149.133
C01255=1132.702,66.266,-53.360,-179.729,6.618,149.134
C01256=1132.706,66.017,-53.343,-179.732,6.618,149.134
C01257=1132.712,65.768,-53.328,-179.734,6.616,149.135
C01258=1132.717,65.518,-53.310,-179.737,6.615,149.135
C01259=1132.722,65.269,-53.294,-179.739,6.614,149.136
C01260=1132.727,65.019,-53.278,-179.743,6.613,149.136
C01261=1132.732,64.770,-53.262,-179.745,6.611,149.137
C01262=1132.737,64.520,-53.246,-179.748,6.610,149.137
C01263=1132.741,64.270,-53.229,-179.750,6.608,149.138
C01264=1132.746,64.022,-53.213,-179.754,6.607,149.138
C01265=1132.751,63.772,-53.197,-179.756,6.606,149.139
C01266=1132.756,63.523,-53.181,-179.758,6.605,149.139
C01267=1132.762,63.273,-53.165,-179.761,6.603,149.140
C01268=1132.766,63.024,-53.148,-179.764,6.602,149.140
C01269=1132.772,62.774,-53.132,-179.767,6.601,149.141
C01270=1132.777,62.525,-53.115,-179.769,6.599,149.141
C01271=1132.782,62.275,-53.100,-179.772,6.598,149.142
C01272=1132.786,62.026,-53.083,-179.775,6.597,149.142
C01273=1132.792,61.776,-53.068,-179.777,6.596,149.143
C01274=1132.796,61.527,-53.051,-179.780,6.594,149.143
C01275=1132.802,61.278,-53.035,-179.782,6.593,149.144
C01276=1132.806,61.028,-53.019,-179.786,6.592,149.144
C01277=1132.812,60.779,-53.003,-179.788,6.590,149.145
C01278=1132.816,60.529,-52.986,-179.791,6.589,149.145
C01279=1132.821,60.280,-52.971,-179.793,6.588,149.146
C01280=1132.827,60.030,-52.955,-179.797,6.586,149.146
C01281=1132.831,59.781,-52.939,-179.799,6.586,149.147
C01282=1132.837,59.531,-52.923,-179.801,6.584,149.147
C01283=1132.841,59.282,-52.906,-179.804,6.582,149.148
C01284=1132.847,59.033,-52.891,-179.807,6.582,149.148
C01285=1132.852,58.783,-52.875,-179.810,6.580,149.149
C01286=1132.856,58.534,-52.859,-179.812,6.579,149.149
C01287=1132.861,58.285,-52.843,-179.815,6.578,149.150
C01288=1132.866,58.035,-52.828,-179.818,6.576,149.150
C01289=1132.871,57.786,-52.811,-179.820,6.575,149.151
C01290=1132.876,57.536,-52.796,-179.823,6.574,149.151
C01291=1132.881,57.286,-52.780,-179.825,6.572,149.152
C01292=1132.886,57.037,-52.763,-179.829,6.571,149.152
C01293=1132.892,56.788,-52.748,-179.831,6.570,149.153
C01294=1132.896,56.538,-52.732,-179.834,6.569,149.153
C01295=1132.901,56.289,-52.716,-179.836,6.568,149.154
C01296=1132.907,56.040,-52.700,-179.839,6.567,149.154
C01297=1132.911,55.790,-52.685,-179.842,6.565,149.155
C01298=1132.916,55.541,-52.669,-179.844,6.564,149.155
C01299=1132.922,55.291,-52.653,-179.847,6.562,149.156
C01300=1132.926,55.042,-52.637,-179.850,6.561,149.156
C01301=1132.932,54.792,-52.621,-179.852,6.560,149.157
C01302=1132.937,54.543,-52.606,-179.855,6.559,149.157
C01303=1132.941,54.293,-52.590,-179.857,6.558,149.158
C01304=1132.946,54.044,-52.575,-179.860,6.557,149.158
C01305=1132.951,53.795,-52.558,-179.863,6.555,149.159
C01306=1132.957,53.525,-52.542,-179.866,6.555,149.159
C01307=1132.962,53.257,-52.525,-179.868,6.553,149.160
C01308=1132.968,52.988,-52.508,-179.871,6.551,149.160
C01309=1132.973,52.720,-52.491,-179.874,6.550,149.161
C01310=1132.978,52.471,-52.476,-179.877,6.548,149.161
C01311=1132.983,52.220,-52.460,-179.879,6.548,149.162
C01312=1132.988,51.971,-52.444,-179.883,6.546,149.162
C01313=1132.994,51.722,-52.428,-179.885,6.545,149.163
C01314=1132.998,51.473,-52.413,-179.887,6.544,149.163
C01315=1133.003,51.223,-52.397,-179.891,6.543,149.164
C01316=1133.008,50.974,-52.381,-179.893,6.542,149.164
C01317=1133.013,50.724,-52.366,-179.896,6.540,149.165
C01318=1133.018,50.475,-52.351,-179.898,6.539,149.165
C01319=1133.023,50.225,-52.335,-179.901,6.538,149.166
C01320=1133.028,49.976,-52.319,-179.904,6.536,149.166
C01321=1133.033,49.727,-52.304,-179.906,6.536,149.167
C01322=1133.038,49.477,-52.289,-179.909,6.534,149.167
C01323=1133.043,49.227,-52.273,-179.911,6.533,149.168
C01324=1133.048,48.978,-52.258,-179.914,6.532,149.168
C01325=1133.053,48.729,-52.242,-179.916,6.531,149.169
C01326=1133.059,48.479,-52.226,-179.919,6.530,149.170
C01327=1133.063,48.230,-52.211,-179.922,6.528,149.170
C01328=1133.068,47.980,-52.195,-179.924,6.527,149.170
C01329=1133.074,47.730,-52.181,-179.927,6.526,149.171
C01330=1133.078,47.481,-52.166,-179.930,6.525,149.172
C01331=1133.084,47.231,-52.150,-179.933,6.524,149.172
C01332=1133.088,46.982,-52.135,-179.935,6.523,149.172
C01333=1133.093,46.732,-52.119,-179.938,6.521,149.173
C01334=1133.099,46.483,-52.103,-179.941,6.520,149.174
C01335=1133.103,46.234,-52.088,-179.943,6.519,149.174
C01336=1133.109,45.984,-52.073,-179.946,6.517,149.174
C01337=1133.113,45.735,-52.058,-179.948,6.517,149.175
C01338=1133.119,45.485,-52.043,-179.951,6.515,149.176
C01339=1133.124,45.235,-52.027,-179.953,6.514,149.176
C01340=1133.128,44.986,-52.012,-179.956,6.513,149.177
C01341=1133.134,44.737,-51.996,-179.959,6.512,149.177
C01342=1133.138,44.488,-51.981,-179.961,6.511,149.178
C01343=1133.144,44.238,-51.967,-179.964,6.509,149.178
C01344=1133.149,43.988,-51.952,-179.967,6.509,149.179
C01345=1133.154,43.739,-51.936,-179.970,6.507,149.179
C01346=1133.158,43.489,-51.921,-179.972,6.506,149.180
C01347=1133.164,43.239,-51.906,-179.975,6.505,149.180
C01348=1133.168,42.990,-51.891,-179.977,6.504,149.181
C01349=1133.174,42.741,-51.875,-179.980,6.503,149.181
C01350=1133.179,42.491,-51.860,-179.983,6.502,149.182
C01351=1133.184,42.242,-51.845,-179.985,6.500,149.182
C01352=1133.189,41.993,-51.830,-179.987,6.500,149.183
C01353=1133.194,41.743,-51.815,-179.990,6.498,149.183
C01354=1133.199,41.493,-51.800,-179.993,6.498,149.184
C01355=1133.205,41.244,-51.785,-179.996,6.496,149.184
C01356=1133.209,40.994,-51.770,-179.998,6.494,149.185
C01357=1133.214,40.744,-51.755,179.999,6.494,149.185
C01358=1133.219,40.495,-51.740,179.996,6.492,149.186
C01359=1133.224,40.246,-51.724,179.994,6.491,149.186
C01360=1133.229,39.996,-51.710,179.991,6.490,149.187
C01361=1133.235,39.747,-51.694,179.989,6.489,149.187
C01362=1133.239,39.498,-51.679,179.986,6.488,149.188
C01363=1133.244,39.248,-51.665,179.984,6.487,149.188
C01364=1133.250,38.998,-51.649,179.980,6.486,149.189
C01365=1133.255,38.749,-51.635,179.978,6.485,149.189
C01366=1133.260,38.499,-51.619,179.976,6.483,149.190
C01367=1133.265,38.250,-51.605,179.973,6.483,149.191
C01368=1133.270,38.001,-51.590,179.970,6.481,149.191
C01369=1133.275,37.751,-51.575,179.968,6.480,149.191
C01370=1133.280,37.501,-51.560,179.965,6.479,149.192
C01371=1133.285,37.252,-51.545,179.963,6.478,149.193
C01372=1133.290,37.002,-51.530,179.960,6.477,149.193
C01373=1133.295,36.753,-51.516,179.958,6.476,149.194
C01374=1133.301,36.503,-51.501,179.954,6.475,149.194
C01375=1133.305,36.254,-51.486,179.952,6.474,149.195
C01376=1133.310,36.004,-51.471,179.949,6.472,149.195
C01377=1133.316,35.755,-51.456,179.947,6.472,149.196
C01378=1133.321,35.505,-51.441,179.944,6.470,149.196
C01379=1133.326,35.256,-51.427,179.942,6.469,149.197
C01380=1133.331,35.006,-51.412,179.939,6.468,149.197
C01381=1133.336,34.756,-51.397,179.936,6.467,149.198
C01382=1133.341,34.507,-51.382,179.934,6.466,149.198
C01383=1133.346,34.258,-51.368,179.931,6.465,149.199
C01384=1133.351,34.008,-51.352,179.929,6.464,149.199
C01385=1133.356,33.759,-51.338,179.926,6.463,149.200
C01386=1133.361,33.509,-51.324,179.924,6.462,149.200
C01387=1133.366,33.259,-51.308,179.921,6.461,149.201
C01388=1133.371,33.010,-51.294,179.919,6.460,149.201
C01389=1133.377,32.761,-51.280,179.916,6.458,149.202
C01390=1133.381,32.512,-51.265,179.913,6.458,149.203
C01391=1133.386,32.262,-51.251,179.910,6.456,149.203
C01392=1133.392,32.012,-51.236,179.908,6.455,149.203
C01393=1133.397,31.763,-51.221,179.905,6.454,149.204
C01394=1133.402,31.513,-51.207,179.903,6.453,149.205
C01395=1133.407,31.263,-51.192,179.900,6.452,149.205
C01396=1133.412,31.014,-51.177,179.897,6.451,149.206
C01397=1133.417,30.764,-51.163,179.895,6.450,149.206
C01398=1133.422,30.515,-51.148,179.892,6.449,149.207
C01399=1133.427,30.265,-51.134,179.890,6.448,149.207
C01400=1133.432,30.016,-51.119,179.887,6.447,149.208
C01401=1133.437,29.767,-51.105,179.885,6.446,149.208
C01402=1133.443,29.517,-51.090,179.882,6.445,149.209
C01403=1133.448,29.267,-51.076,179.879,6.444,149.209
C01404=1133.452,29.018,-51.061,179.877,6.442,149.210
C01405=1133.457,28.768,-51.047,179.874,6.441,149.210
C01406=1133.462,28.518,-51.032,179.872,6.441,149.211
C01407=1133.468,28.269,-51.019,179.869,6.439,149.211
C01408=1133.473,28.020,-51.004,179.867,6.438,149.212
C01409=1133.478,27.770,-50.990,179.864,6.437,149.213
C01410=1133.484,27.501,-50.974,179.861,6.436,149.213
C01411=1133.489,27.232,-50.958,179.858,6.435,149.214
C01412=1133.494,26.963,-50.943,179.855,6.434,149.214
C01413=1133.499,26.694,-50.927,179.853,6.433,149.215
C01414=1133.505,26.445,-50.913,179.850,6.431,149.215
C01415=1133.510,26.195,-50.899,179.848,6.431,149.216
C01416=1133.515,25.945,-50.884,179.845,6.430,149.216
C01417=1133.520,25.695,-50.870,179.842,6.429,149.217
C01418=1133.525,25.446,-50.856,179.840,6.428,149.217
C01419=1133.531,25.197,-50.842,179.837,6.427,149.218
C01420=1133.536,24.947,-50.827,179.835,6.426,149.218
C01421=1133.541,24.698,-50.812,179.833,6.425,149.219
C01422=1133.545,24.448,-50.798,179.829,6.424,149.220
C01423=1133.550,24.199,-50.784,179.827,6.423,149.220
C01424=1133.556,23.950,-50.770,179.824,6.421,149.220
C01425=1133.561,23.700,-50.756,179.822,6.421,149.221
C01426=1133.566,23.450,-50.741,179.820,6.420,149.222
C01427=1133.571,23.200,-50.727,179.817,6.418,149.222
C01428=1133.576,22.951,-50.713,179.814,6.418,149.223
C01429=1133.581,22.702,-50.699,179.811,6.416,149.223
C01430=1133.586,22.452,-50.685,179.809,6.416,149.224
C01431=1133.591,22.202,-50.670,179.807,6.415,149.224
C01432=1133.597,21.953,-50.657,179.804,6.413,149.225
C01433=1133.602,21.703,-50.643,179.802,6.413,149.225
C01434=1133.607,21.453,-50.629,179.798,6.411,149.226
C01435=1133.611,21.204,-50.615,179.796,6.411,149.226
C01436=1133.617,20.955,-50.601,179.794,6.410,149.227
C01437=1133.622,20.705,-50.587,179.791,6.409,149.228
C01438=1133.627,20.455,-50.573,179.789,6.408,149.228
C01439=1133.632,20.206,-50.558,179.787,6.407,149.228
C01440=1133.637,19.957,-50.544,179.783,6.406,149.229
C01441=1133.642,19.707,-50.530,179.781,6.405,149.230
C01442=1133.647,19.457,-50.517,179.778,6.403,149.230
C01443=1133.653,19.208,-50.503,179.776,6.403,149.231
C01444=1133.658,18.958,-50.488,179.774,6.402,149.231
C01445=1133.663,18.708,-50.474,179.771,6.400,149.232
C01446=1133.668,18.459,-50.461,179.768,6.400,149.232
C01447=1133.673,18.210,-50.446,179.766,6.399,149.233
C01448=1133.678,17.959,-50.433,179.763,6.398,149.233
C01449=1133.684,17.710,-50.419,179.760,6.397,149.234
C01450=1133.688,17.461,-50.405,179.758,6.396,149.234
C01451=1133.693,17.211,-50.390,179.756,6.395,149.235
C01452=1133.698,16.962,-50.377,179.753,6.394,149.236
C01453=1133.704,16.712,-50.364,179.750,6.393,149.236
C01454=1133.708,16.462,-50.349,179.748,6.392,149.236
C01455=1133.714,16.213,-50.335,179.745,6.391,149.237
C01456=1133.719,15.964,-50.321,179.743,6.390,149.238
C01457=1133.724,15.713,-50.308,179.740,6.389,149.238
C01458=1133.729,15.465,-50.294,179.738,6.388,149.239
C01459=1133.734,15.215,-50.280,179.735,6.387,149.239
C01460=1133.740,14.965,-50.267,179.733,6.386,149.240
C01461=1133.745,14.715,-50.252,179.731,6.385,149.240
C01462=1133.749,14.466,-50.239,179.727,6.384,149.241
C01463=1133.755,14.216,-50.226,179.725,6.383,149.241
C01464=1133.760,13.967,-50.211,179.723,6.383,149.242
C01465=1133.765,13.717,-50.197,179.720,6.381,149.242
C01466=1133.770,13.468,-50.184,179.718,6.381,149.243
C01467=1133.775,13.218,-50.170,179.715,6.380,149.243
C01468=1133.780,12.969,-50.156,179.712,6.378,149.244
C01469=1133.786,12.719,-50.143,179.710,6.378,149.244
C01470=1133.791,12.470,-50.129,179.708,6.377,149.245
C01471=1133.796,12.220,-50.116,179.705,6.376,149.246
C01472=1133.801,11.970,-50.102,179.702,6.375,149.246
C01473=1133.806,11.721,-50.088,179.700,6.374,149.247
C01474=1133.811,11.471,-50.075,179.698,6.374,149.247
C01475=1133.816,11.222,-50.061,179.695,6.372,149.248
C01476=1133.822,10.972,-50.047,179.692,6.372,149.248
C01477=1133.826,10.723,-50.034,179.690,6.371,149.249
C01478=1133.832,10.473,-50.020,179.687,6.369,149.249
C01479=1133.837,10.224,-50.006,179.684,6.369,149.250
C01480=1133.842,9.973,-49.993,179.682,6.368,149.250
C01481=1133.847,9.724,-49.979,179.680,6.366,149.251
C01482=1133.852,9.474,-49.967,179.677,6.366,149.252
C01483=1133.857,9.225,-49.952,179.675,6.365,149.252
C01484=1133.863,8.975,-49.939,179.672,6.363,149.253
C01485=1133.867,8.726,-49.925,179.669,6.363,149.253
C01486=1133.873,8.476,-49.912,179.667,6.362,149.254
C01487=1133.878,8.226,-49.898,179.665,6.361,149.254
C01488=1133.883,7.977,-49.885,179.662,6.360,149.255
C01489=1133.888,7.727,-49.871,179.659,6.359,149.255
C01490=1133.893,7.478,-49.858,179.657,6.359,149.256
C01491=1133.898,7.228,-49.845,179.654,6.357,149.256
C01492=1133.904,6.979,-49.831,179.652,6.357,149.257
C01493=1133.908,6.729,-49.818,179.650,6.356,149.257
C01494=1133.914,6.480,-49.804,179.647,6.355,149.258
C01495=1133.918,6.230,-49.791,179.644,6.354,149.259
C01496=1133.924,5.980,-49.778,179.642,6.353,149.259
C01497=1133.928,5.731,-49.764,179.639,6.353,149.260
C01498=1133.934,5.481,-49.751,179.637,6.352,149.260
C01499=1133.939,5.232,-49.738,179.634,6.350,149.261
C01500=1133.944,4.982,-49.724,179.632,6.350,149.261
C01501=1133.949,4.733,-49.712,179.630,6.349,149.262
C01502=1133.955,4.482,-49.698,179.627,6.347,149.262
C01503=1133.960,4.233,-49.684,179.624,6.347,149.263
C01504=1133.965,3.983,-49.671,179.622,6.346,149.263
C01505=1133.971,3.734,-49.658,179.620,6.345,149.264
C01506=1133.975,3.484,-49.644,179.617,6.344,149.265
C01507=1133.980,3.235,-49.632,179.614,6.343,149.265
C01508=1133.986,2.985,-49.618,179.612,6.342,149.265
C01509=1133.990,2.735,-49.605,179.610,6.342,149.266
C01510=1133.996,2.486,-49.592,179.607,6.340,149.267
C01511=1134.000,2.236,-49.579,179.605,6.340,149.267
C01512=1134.006,1.987,-49.565,179.602,6.339,149.268
C01513=1134.011,1.737,-49.553,179.600,6.338,149.268
C01514=1134.017,1.468,-49.538,179.597,6.337,149.269
C01515=1134.023,1.198,-49.524,179.594,6.336,149.269
C01516=1134.028,0.928,-49.510,179.591,6.335,149.270
C01517=1134.034,0.659,-49.495,179.589,6.334,149.271
C01518=1134.038,0.409,-49.482,179.587,6.334,149.271
C01519=1134.044,0.160,-49.469,179.584,6.332,149.272
C01520=1134.049,-0.090,-49.456,179.581,6.332,149.272
C01521=1134.054,-0.340,-49.444,179.579,6.331,149.273
C01522=1134.059,-0.589,-49.430,179.577,6.330,149.273
C01523=1134.064,-0.838,-49.417,179.574,6.330,149.274
C01524=1134.070,-1.088,-49.403,179.572,6.328,149.274
C01525=1134.075,-1.338,-49.391,179.569,6.328,149.275
C01526=1134.080,-1.587,-49.378,179.567,6.327,149.275
C01527=1134.085,-1.837,-49.365,179.565,6.326,149.276
C01528=1134.090,-2.086,-49.352,179.561,6.325,149.277
C01529=1134.095,-2.336,-49.339,179.559,6.324,149.277
C01530=1134.101,-2.586,-49.326,179.557,6.323,149.277
C01531=1134.106,-2.835,-49.313,179.554,6.323,149.278
C01532=1134.112,-3.085,-49.300,179.552,6.322,149.279
C01533=1134.116,-3.334,-49.286,179.549,6.320,149.279
C01534=1134.121,-3.584,-49.274,179.547,6.320,149.280
C01535=1134.126,-3.833,-49.261,179.544,6.319,149.280
C01536=1134.131,-4.083,-49.248,179.542,6.318,149.281
C01537=1134.136,-4.333,-49.235,179.539,6.317,149.281
C01538=1134.142,-4.582,-49.222,179.537,6.316,149.282
C01539=1134.147,-4.832,-49.209,179.535,6.315,149.282
C01540=1134.152,-5.082,-49.196,179.532,6.315,149.283
C01541=1134.157,-5.331,-49.184,179.530,6.314,149.283
C01542=1134.162,-5.580,-49.171,179.527,6.313,149.284
C01543=1134.168,-5.831,-49.158,179.524,6.312,149.285
C01544=1134.173,-6.081,-49.146,179.522,6.311,149.285
C01545=1134.178,-6.330,-49.133,179.520,6.311,149.286
C01546=1134.184,-6.580,-49.120,179.517,6.310,149.286
C01547=1134.188,-6.830,-49.107,179.515,6.309,149.287
C01548=1134.194,-7.079,-49.094,179.512,6.308,149.287
C01549=1134.199,-7.328,-49.082,179.510,6.307,149.288
C01550=1134.204,-7.578,-49.069,179.508,6.307,149.288
C01551=1134.209,-7.828,-49.056,179.505,6.306,149.289
C01552=1134.214,-8.077,-49.043,179.503,6.305,149.290
C01553=1134.219,-8.327,-49.030,179.500,6.304,149.290
C01554=1134.224,-8.576,-49.018,179.498,6.303,149.290
C01555=1134.229,-8.826,-49.005,179.495,6.303,149.291
C01556=1134.235,-9.076,-48.992,179.493,6.302,149.292
C01557=1134.240,-9.325,-48.980,179.491,6.301,149.292
C01558=1134.245,-9.575,-48.967,179.488,6.301,149.293
C01559=1134.250,-9.825,-48.954,179.485,6.299,149.293
C01560=1134.255,-10.074,-48.942,179.483,6.298,149.294
C01561=1134.260,-10.324,-48.930,179.480,6.298,149.294
C01562=1134.266,-10.574,-48.916,179.478,6.297,149.295
C01563=1134.271,-10.823,-48.904,179.476,6.296,149.295
C01564=1134.276,-11.073,-48.891,179.473,6.296,149.296
C01565=1134.281,-11.322,-48.878,179.471,6.294,149.297
C01566=1134.287,-11.572,-48.866,179.468,6.293,149.297
C01567=1134.292,-11.822,-48.854,179.466,6.293,149.298
C01568=1134.297,-12.071,-48.841,179.464,6.292,149.298
C01569=1134.302,-12.320,-48.829,179.461,6.291,149.299
C01570=1134.307,-12.571,-48.816,179.459,6.291,149.299
C01571=1134.313,-12.820,-48.803,179.456,6.289,149.300
C01572=1134.318,-13.070,-48.791,179.454,6.289,149.300
C01573=1134.323,-13.320,-48.779,179.451,6.288,149.301
C01574=1134.328,-13.569,-48.766,179.449,6.287,149.301
C01575=1134.333,-13.818,-48.753,179.447,6.287,149.302
C01576=1134.338,-14.068,-48.740,179.444,6.286,149.303
C01577=1134.343,-14.318,-48.729,179.442,6.285,149.303
C01578=1134.348,-14.568,-48.716,179.439,6.284,149.304
C01579=1134.354,-14.817,-48.703,179.437,6.283,149.304
C01580=1134.359,-15.067,-48.692,179.434,6.283,149.305
C01581=1134.364,-15.316,-48.679,179.432,6.282,149.305
C01582=1134.370,-15.566,-48.667,179.430,6.281,149.306
C01583=1134.375,-15.815,-48.654,179.427,6.281,149.306
C01584=1134.379,-16.065,-48.641,179.425,6.280,149.307
C01585=1134.385,-16.315,-48.630,179.423,6.279,149.307
C01586=1134.390,-16.565,-48.617,179.420,6.278,149.308
C01587=1134.395,-16.815,-48.605,179.418,6.277,149.308
C01588=1134.400,-17.064,-48.592,179.415,6.277,149.309
C01589=1134.405,-17.313,-48.580,179.413,6.276,149.310
C01590=1134.411,-17.563,-48.568,179.411,6.275,149.310
C01591=1134.416,-17.813,-48.555,179.408,6.275,149.311
C01592=1134.421,-18.062,-48.544,179.406,6.274,149.311
C01593=1134.427,-18.312,-48.531,179.403,6.273,149.312
C01594=1134.432,-18.562,-48.519,179.400,6.272,149.312
C01595=1134.437,-18.812,-48.506,179.398,6.271,149.313
C01596=1134.442,-19.062,-48.494,179.396,6.270,149.313
C01597=1134.447,-19.311,-48.482,179.393,6.270,149.314
C01598=1134.452,-19.561,-48.470,179.391,6.269,149.315
C01599=1134.458,-19.810,-48.457,179.389,6.268,149.315
C01600=1134.463,-20.060,-48.445,179.386,6.268,149.316
C01601=1134.468,-20.309,-48.433,179.384,6.267,149.316
C01602=1134.474,-20.559,-48.421,179.382,6.266,149.317
C01603=1134.479,-20.809,-48.408,179.379,6.265,149.317
C01604=1134.484,-21.059,-48.396,179.376,6.264,149.318
C01605=1134.489,-21.308,-48.384,179.374,6.264,149.318
C01606=1134.494,-21.558,-48.372,179.371,6.263,149.319
C01607=1134.499,-21.807,-48.360,179.369,6.262,149.319
C01608=1134.505,-22.057,-48.348,179.367,6.262,149.320
C01609=1134.510,-22.307,-48.336,179.364,6.261,149.321
C01610=1134.515,-22.556,-48.323,179.362,6.260,149.321
C01611=1134.521,-22.806,-48.311,179.360,6.260,149.322
C01612=1134.526,-23.055,-48.299,179.357,6.259,149.322
C01613=1134.530,-23.305,-48.288,179.355,6.258,149.323
C01614=1134.536,-23.555,-48.276,179.353,6.258,149.323
C01615=1134.541,-23.804,-48.263,179.350,6.256,149.324
C01616=1134.546,-24.054,-48.251,179.348,6.256,149.324
C01617=1134.552,-24.304,-48.239,179.345,6.255,149.325
C01618=1134.557,-24.575,-48.226,179.343,6.255,149.326
C01619=1134.563,-24.844,-48.214,179.341,6.254,149.326
C01620=1134.568,-25.115,-48.201,179.338,6.253,149.327
C01621=1134.574,-25.384,-48.187,179.335,6.252,149.327
C01622=1134.579,-25.633,-48.176,179.333,6.251,149.328
C01623=1134.585,-25.883,-48.164,179.330,6.251,149.328
C01624=1134.590,-26.133,-48.152,179.328,6.250,149.329
C01625=1134.595,-26.383,-48.139,179.326,6.249,149.329
C01626=1134.600,-26.632,-48.128,179.323,6.249,149.330
C01627=1134.605,-26.882,-48.116,179.321,6.248,149.330
C01628=1134.611,-27.132,-48.104,179.319,6.247,149.331
C01629=1134.616,-27.381,-48.092,179.316,6.247,149.332
C01630=1134.621,-27.631,-48.080,179.314,6.246,149.332
C01631=1134.626,-27.881,-48.068,179.312,6.245,149.333
C01632=1134.632,-28.131,-48.057,179.309,6.245,149.333
C01633=1134.637,-28.380,-48.044,179.307,6.244,149.334
C01634=1134.641,-28.630,-48.033,179.305,6.243,149.334
C01635=1134.647,-28.880,-48.021,179.302,6.243,149.335
C01636=1134.653,-29.129,-48.009,179.299,6.241,149.335
C01637=1134.657,-29.379,-47.998,179.297,6.240,149.336
C01638=1134.663,-29.628,-47.985,179.295,6.240,149.337
C01639=1134.668,-29.878,-47.973,179.292,6.239,149.337
C01640=1134.673,-30.128,-47.962,179.290,6.238,149.338
C01641=1134.678,-30.378,-47.950,179.288,6.238,149.338
C01642=1134.684,-30.627,-47.938,179.285,6.237,149.339
C01643=1134.689,-30.877,-47.926,179.283,6.236,149.339
C01644=1134.694,-31.127,-47.915,179.281,6.236,149.340
C01645=1134.699,-31.376,-47.903,179.278,6.235,149.340
C01646=1134.704,-31.625,-47.892,179.276,6.234,149.341
C01647=1134.710,-31.875,-47.880,179.274,6.234,149.341
C01648=1134.715,-32.125,-47.868,179.271,6.233,149.342
C01649=1134.720,-32.375,-47.857,179.269,6.232,149.342
C01650=1134.725,-32.625,-47.845,179.267,6.232,149.343
C01651=1134.731,-32.875,-47.833,179.264,6.231,149.344
C01652=1134.736,-33.124,-47.822,179.262,6.230,149.344
C01653=1134.741,-33.374,-47.810,179.260,6.230,149.345
C01654=1134.747,-33.623,-47.798,179.258,6.229,149.345
C01655=1134.751,-33.873,-47.787,179.255,6.229,149.346
C01656=1134.757,-34.123,-47.775,179.253,6.228,149.346
C01657=1134.761,-34.373,-47.764,179.251,6.227,149.347
C01658=1134.768,-34.622,-47.752,179.248,6.227,149.347
C01659=1134.773,-34.872,-47.740,179.246,6.226,149.348
C01660=1134.778,-35.121,-47.729,179.244,6.225,149.348
C01661=1134.783,-35.371,-47.717,179.241,6.225,149.349
C01662=1134.788,-35.621,-47.706,179.239,6.224,149.350
C01663=1134.794,-35.870,-47.694,179.237,6.223,149.350
C01664=1134.798,-36.120,-47.683,179.234,6.223,149.351
C01665=1134.804,-36.370,-47.671,179.232,6.222,149.351
C01666=1134.809,-36.619,-47.660,179.229,6.221,149.352
C01667=1134.814,-36.869,-47.648,179.227,6.220,149.352
C01668=1134.820,-37.119,-47.636,179.225,6.220,149.353
C01669=1134.825,-37.368,-47.625,179.222,6.219,149.353
C01670=1134.830,-37.618,-47.613,179.220,6.218,149.354
C01671=1134.835,-37.868,-47.602,179.218,6.218,149.354
C01672=1134.841,-38.117,-47.590,179.215,6.217,149.355
C01673=1134.846,-38.367,-47.579,179.213,6.216,149.355
C01674=1134.851,-38.617,-47.568,179.211,6.216,149.356
C01675=1134.856,-38.867,-47.557,179.208,6.215,149.357
C01676=1134.862,-39.116,-47.545,179.206,6.214,149.357
C01677=1134.867,-39.366,-47.534,179.204,6.214,149.358
C01678=1134.872,-39.616,-47.522,179.201,6.213,149.358
C01679=1134.877,-39.865,-47.511,179.199,6.213,149.359
C01680=1134.883,-40.114,-47.499,179.197,6.212,149.359
C01681=1134.888,-40.365,-47.489,179.194,6.211,149.360
C01682=1134.893,-40.615,-47.477,179.192,6.211,149.360
C01683=1134.898,-40.864,-47.465,179.190,6.210,149.361
C01684=1134.903,-41.113,-47.455,179.188,6.209,149.361
C01685=1134.909,-41.363,-47.443,179.185,6.209,149.362
C01686=1134.914,-41.613,-47.432,179.183,6.208,149.363
C01687=1134.920,-41.863,-47.421,179.181,6.207,149.363
C01688=1134.924,-42.112,-47.409,179.178,6.207,149.364
C01689=1134.930,-42.362,-47.397,179.176,6.206,149.364
C01690=1134.935,-42.612,-47.387,179.174,6.205,149.365
C01691=1134.940,-42.861,-47.376,179.171,6.204,149.365
C01692=1134.946,-43.111,-47.364,179.169,6.204,149.366
C01693=1134.950,-43.361,-47.353,179.167,6.203,149.366
C01694=1134.957,-43.611,-47.342,179.164,6.202,149.367
C01695=1134.961,-43.860,-47.331,179.162,6.203,149.367
C01696=1134.966,-44.110,-47.319,179.160,6.202,149.368
C01697=1134.972,-44.359,-47.308,179.158,6.201,149.368
C01698=1134.977,-44.610,-47.297,179.156,6.200,149.369
C01699=1134.982,-44.859,-47.286,179.153,6.200,149.370
C01700=1134.988,-45.108,-47.274,179.151,6.199,149.370
C01701=1134.993,-45.359,-47.264,179.149,6.199,149.371
C01702=1134.997,-45.608,-47.253,179.146,6.198,149.371
C01703=1135.003,-45.857,-47.241,179.144,6.197,149.372
C01704=1135.008,-46.108,-47.230,179.142,6.197,149.372
C01705=1135.014,-46.358,-47.219,179.139,6.196,149.373
C01706=1135.019,-46.607,-47.208,179.137,6.195,149.373
C01707=1135.024,-46.857,-47.197,179.135,6.195,149.374
C01708=1135.030,-47.106,-47.186,179.132,6.194,149.374
C01709=1135.035,-47.356,-47.175,179.130,6.194,149.375
C01710=1135.040,-47.606,-47.164,179.128,6.193,149.376
C01711=1135.045,-47.855,-47.153,179.125,6.192,149.376
C01712=1135.051,-48.105,-47.142,179.124,6.192,149.377
C01713=1135.056,-48.355,-47.130,179.121,6.192,149.377
C01714=1135.061,-48.605,-47.120,179.119,6.191,149.378
C01715=1135.067,-48.855,-47.108,179.117,6.190,149.378
C01716=1135.072,-49.103,-47.097,179.114,6.190,149.379
C01717=1135.077,-49.354,-47.087,179.112,6.189,149.379
C01718=1135.082,-49.603,-47.075,179.110,6.188,149.380
C01719=1135.088,-49.853,-47.065,179.108,6.187,149.380
C01720=1135.093,-50.103,-47.053,179.105,6.187,149.381
C01721=1135.098,-50.352,-47.043,179.103,6.186,149.381
C01722=1135.104,-50.623,-47.031,179.100,6.185,149.382
C01723=1135.110,-50.894,-47.019,179.098,6.185,149.383
C01724=1135.115,-51.164,-47.007,179.096,6.184,149.383
C01725=1135.121,-51.436,-46.996,179.093,6.184,149.384
C01726=1135.126,-51.685,-46.985,179.091,6.183,149.384
C01727=1135.132,-51.935,-46.974,179.089,6.182,149.385
C01728=1135.137,-52.185,-46.962,179.086,6.182,149.386
C01729=1135.142,-52.435,-46.952,179.084,6.181,149.386
C01730=1135.147,-52.684,-46.941,179.081,6.180,149.386
C01731=1135.153,-52.934,-46.931,179.080,6.180,149.387
C01732=1135.157,-53.183,-46.919,179.077,6.180,149.388
C01733=1135.164,-53.433,-46.909,179.075,6.179,149.388
C01734=1135.169,-53.683,-46.898,179.073,6.179,149.389
C01735=1135.174,-53.932,-46.887,179.071,6.178,149.389
C01736=1135.179,-54.183,-46.877,179.068,6.177,149.390
C01737=1135.184,-54.431,-46.866,179.066,6.177,149.390
C01738=1135.189,-54.682,-46.855,179.064,6.176,149.391
C01739=1135.195,-54.932,-46.844,179.061,6.175,149.391
C01740=1135.200,-55.181,-46.833,179.059,6.175,149.392
C01741=1135.205,-55.431,-46.822,179.057,6.175,149.392
C01742=1135.210,-55.680,-46.811,179.055,6.174,149.393
C01743=1135.215,-55.931,-46.801,179.053,6.173,149.393
C01744=1135.221,-56.180,-46.791,179.050,6.173,149.394
C01745=1135.226,-56.430,-46.779,179.048,6.172,149.395
C01746=1135.231,-56.679,-46.769,179.046,6.171,149.395
C01747=1135.236,-56.930,-46.759,179.044,6.170,149.396
C01748=1135.242,-57.179,-46.748,179.041,6.170,149.396
C01749=1135.247,-57.429,-46.736,179.039,6.170,149.397
C01750=1135.253,-57.679,-46.726,179.037,6.169,149.397
C01751=1135.258,-57.928,-46.715,179.035,6.169,149.398
C01752=1135.263,-58.178,-46.705,179.032,6.168,149.398
C01753=1135.269,-58.427,-46.695,179.030,6.167,149.399
C01754=1135.274,-58.678,-46.684,179.028,6.167,149.399
C01755=1135.279,-58.926,-46.673,179.026,6.166,149.400
C01756=1135.284,-59.177,-46.662,179.023,6.165,149.401
C01757=1135.290,-59.426,-46.652,179.021,6.166,149.401
C01758=1135.295,-59.677,-46.642,179.019,6.165,149.401
C01759=1135.300,-59.925,-46.631,179.017,6.164,149.402
C01760=1135.305,-60.176,-46.620,179.014,6.164,149.403
C01761=1135.311,-60.425,-46.610,179.012,6.163,149.403
C01762=1135.316,-60.675,-46.599,179.010,6.162,149.404
C01763=1135.321,-60.924,-46.589,179.008,6.161,149.404
C01764=1135.327,-61.174,-46.578,179.006,6.162,149.405
C01765=1135.332,-61.424,-46.568,179.004,6.161,149.405
C01766=1135.337,-61.674,-46.558,179.001,6.160,149.406
C01767=1135.342,-61.924,-46.547,178.999,6.159,149.406
C01768=1135.348,-62.174,-46.537,178.996,6.159,149.407
C01769=1135.352,-62.423,-46.525,178.994,6.158,149.407
C01770=1135.358,-62.673,-46.515,178.993,6.158,149.408
C01771=1135.364,-62.922,-46.505,178.991,6.158,149.408
C01772=1135.369,-63.172,-46.494,178.988,6.157,149.409
C01773=1135.374,-63.422,-46.484,178.986,6.156,149.410
C01774=1135.379,-63.672,-46.474,178.983,6.156,149.410
C01775=1135.385,-63.922,-46.463,178.981,6.155,149.411
C01776=1135.390,-64.171,-46.453,178.979,6.154,149.411
C01777=1135.395,-64.421,-46.442,178.977,6.154,149.412
C01778=1135.401,-64.671,-46.432,178.975,6.154,149.412
C01779=1135.406,-64.920,-46.422,178.973,6.153,149.413
C01780=1135.411,-65.170,-46.412,178.970,6.152,149.413
C01781=1135.416,-65.420,-46.401,178.968,6.152,149.414
C01782=1135.421,-65.670,-46.391,178.966,6.152,149.414
C01783=1135.427,-65.919,-46.381,178.964,6.151,149.415
C01784=1135.432,-66.169,-46.370,178.962,6.150,149.415
C01785=1135.437,-66.419,-46.360,178.959,6.150,149.416
C01786=1135.443,-66.669,-46.350,178.957,6.149,149.417
C01787=1135.449,-66.918,-46.339,178.955,6.148,149.417
C01788=1135.454,-67.168,-46.329,178.953,6.148,149.417
C01789=1135.458,-67.418,-46.319,178.951,6.148,149.418
C01790=1135.464,-67.667,-46.309,178.948,6.147,149.419
C01791=1135.469,-67.917,-46.298,178.946,6.147,149.419
C01792=1135.475,-68.167,-46.288,178.944,6.146,149.420
C01793=1135.480,-68.417,-46.278,178.942,6.146,149.420
C01794=1135.485,-68.667,-46.267,178.940,6.145,149.421
C01795=1135.491,-68.916,-46.257,178.937,6.145,149.421
C01796=1135.496,-69.166,-46.248,178.935,6.144,149.422
C01797=1135.501,-69.416,-46.237,178.933,6.143,149.422
C01798=1135.506,-69.665,-46.227,178.931,6.142,149.423
C01799=1135.512,-69.915,-46.217,178.929,6.143,149.423
C01800=1135.517,-70.164,-46.206,178.927,6.142,149.424
C01801=1135.522,-70.415,-46.196,178.924,6.141,149.424
C01802=1135.527,-70.664,-46.186,178.922,6.140,149.425
C01803=1135.533,-70.913,-46.176,178.920,6.140,149.425
C01804=1135.538,-71.164,-46.165,178.918,6.140,149.426
C01805=1135.543,-71.413,-46.155,178.916,6.139,149.427
C01806=1135.549,-71.663,-46.146,178.914,6.139,149.427
C01807=1135.554,-71.913,-46.136,178.911,6.138,149.428
C01808=1135.559,-72.163,-46.126,178.909,6.138,149.428
C01809=1135.565,-72.412,-46.115,178.907,6.138,149.429
C01810=1135.570,-72.662,-46.105,178.905,6.137,149.429
C01811=1135.576,-72.912,-46.095,178.903,6.136,149.430
C01812=1135.580,-73.161,-46.085,178.900,6.135,149.430
C01813=1135.586,-73.412,-46.075,178.898,6.136,149.431
C01814=1135.592,-73.661,-46.065,178.896,6.135,149.431
C01815=1135.597,-73.911,-46.055,178.894,6.134,149.432
C01816=1135.602,-74.161,-46.045,178.892,6.133,149.432
C01817=1135.607,-74.410,-46.035,178.890,6.133,149.433
